            IF (_MessageLevel > E_MessageType.eMessageError)
            THEN
              _stMsg.eType                                    := E_MessageType.eMessageInfo;
              _stMsg.eSubdevice                               := e_Subdevice.Application_Finish;
              _stMsg.iErrorNumber                             := 0;
              _stMsg.sText                                    := concat(TO_STRING(E_INSTANCE.OUTFEED_ROBOT_R1), ': _wDisable ');
              _stMsg.sText                                    := concat(_stMsg.sText, _ItfProcessCollector[E_INSTANCE.OUTFEED_ROBOT_R1].BitsToString(_wDisable));
              f_MessageSet(_stMsg);
            END_IF
          END_IF
        ELSE
          _InstanceCtrl[E_INSTANCE.OUTFEED_ROBOT_R1].Cmd      := E_INSTANCE_CMD.ENABLE;
        END_IF
      END_CASE

      E_INSTANCE_STATE.ENABLED:
        CASE _InstanceState[E_INSTANCE.OUTFEED_ROBOT_R1].Progress
        OF
          E_PROGRESS.PROGRESS_OCCUPIED:
            _InstanceCtrl[E_INSTANCE.OUTFEED_ROBOT_R1].Cmd    := E_INSTANCE_CMD.PROCEED;
        END_CASE


      E_INSTANCE_STATE.WORKING:
        CASE _InstanceState[E_INSTANCE.OUTFEED_ROBOT_R1].Progress
        OF
          E_PROGRESS.PROGRESS_BUSY:
            _tonProcess [E_INSTANCE.OUTFEED_ROBOT_R1]
                                                  (IN         := FALSE, 
                                                   PT         := _tProcess[E_INSTANCE.OUTFEED_ROBOT_R1]);

            _InstanceCtrl[E_INSTANCE.OUTFEED_ROBOT_R1].Cmd    := E_INSTANCE_CMD.WORK;
    

          E_PROGRESS.PROGRESS_CHECK:
            _tonProcess [E_INSTANCE.OUTFEED_ROBOT_R1]
                                                  (IN         := TRUE, 
                                                   PT         := _tProcess[E_INSTANCE.OUTFEED_ROBOT_R1]);
    
            IF _tonProcess [E_INSTANCE.OUTFEED_ROBOT_R1].Q
            THEN
              _InstanceCtrl[E_INSTANCE.OUTFEED_ROBOT_R1].Cmd  := E_INSTANCE_CMD.FINISH;
            END_IF
        END_CASE

      E_INSTANCE_STATE.FINISH:
        CASE _InstanceState[E_INSTANCE.OUTFEED_ROBOT_R1].Progress
        OF
          E_PROGRESS.PROGRESS_BUSY:
            _InstanceCtrl[E_INSTANCE.OUTFEED_ROBOT_R1].Cmd    := E_INSTANCE_CMD.FINISH;

          E_PROGRESS.PROGRESS_DONE:
            _InstanceCtrl[E_INSTANCE.OUTFEED_ROBOT_R1].Cmd    := E_INSTANCE_CMD.DISABLE;
        END_CASE
      END_CASE

    //-------------------------------------------------------------------------
    // E_INSTANCE.OUTFEED_ROBOT_R2
    //-------------------------------------------------------------------------
    CASE _InstanceState[E_INSTANCE.OUTFEED_ROBOT_R2].State
    OF
    E_INSTANCE_STATE.DISABLED:
      CASE _InstanceState[E_INSTANCE.OUTFEED_ROBOT_R2].Progress
      OF
      E_PROGRESS.PROGRESS_BUSY:
        IF (_ItfProcessCollector[E_INSTANCE.OUTFEED_ROBOT_R2].QueueProcessCount < 12)
        THEN
          _InstanceCtrl[E_INSTANCE.OUTFEED_ROBOT_R2].Cmd      := E_INSTANCE_CMD.DISABLE;

          IF NOT (_ItfProcessCollector[E_INSTANCE.OUTFEED_ROBOT_R2].BitGet(_wDisable, TO_BYTE(E_INSTANCE.OUTFEED_ROBOT_R2-1)))
          THEN
            _wDisable                                         := _ItfProcessCollector[E_INSTANCE.OUTFEED_ROBOT_R2].
                                                                 BitSet(_wDisable, TO_BYTE(E_INSTANCE.OUTFEED_ROBOT_R2-1));

            IF (_MessageLevel > E_MessageType.eMessageError)
            THEN
              _stMsg.eType                                    := E_MessageType.eMessageInfo;
              _stMsg.eSubdevice                               := e_Subdevice.Application_Finish;
              _stMsg.iErrorNumber                             := 0;
              _stMsg.sText                                    := concat(TO_STRING(E_INSTANCE.OUTFEED_ROBOT_R2), ': _wDisable ');
              _stMsg.sText                                    := concat(_stMsg.sText, _ItfProcessCollector[E_INSTANCE.OUTFEED_ROBOT_R2].BitsToString(_wDisable));
              f_MessageSet(_stMsg);
            END_IF
          END_IF
        ELSE
          _InstanceCtrl[E_INSTANCE.OUTFEED_ROBOT_R2].Cmd      := E_INSTANCE_CMD.ENABLE;
        END_IF
      END_CASE

      E_INSTANCE_STATE.ENABLED:
        CASE _InstanceState[E_INSTANCE.OUTFEED_ROBOT_R2].Progress
        OF
          E_PROGRESS.PROGRESS_OCCUPIED:
            _InstanceCtrl[E_INSTANCE.OUTFEED_ROBOT_R2].Cmd    := E_INSTANCE_CMD.PROCEED;
        END_CASE

      E_INSTANCE_STATE.WORKING:
        CASE _InstanceState[E_INSTANCE.OUTFEED_ROBOT_R2].Progress
        OF
          E_PROGRESS.PROGRESS_BUSY:
            _tonProcess [E_INSTANCE.OUTFEED_ROBOT_R2]
                                                  (IN         := FALSE, 
                                                   PT         := _tProcess[E_INSTANCE.OUTFEED_ROBOT_R2]);

            _InstanceCtrl[E_INSTANCE.OUTFEED_ROBOT_R2].Cmd    := E_INSTANCE_CMD.WORK;

    
          E_PROGRESS.PROGRESS_CHECK:
            _tonProcess [E_INSTANCE.OUTFEED_ROBOT_R2]
                                                  (IN         := TRUE, 
                                                   PT         := _tProcess[E_INSTANCE.OUTFEED_ROBOT_R2]);
    
            IF _tonProcess [E_INSTANCE.OUTFEED_ROBOT_R2].Q
            THEN
              _InstanceCtrl[E_INSTANCE.OUTFEED_ROBOT_R2].Cmd  := E_INSTANCE_CMD.FINISH;
            END_IF
        END_CASE

      E_INSTANCE_STATE.FINISH:
        CASE _InstanceState[E_INSTANCE.OUTFEED_ROBOT_R2].Progress
        OF
          E_PROGRESS.PROGRESS_BUSY:
            _InstanceCtrl[E_INSTANCE.OUTFEED_ROBOT_R2].Cmd    := E_INSTANCE_CMD.FINISH;

          E_PROGRESS.PROGRESS_DONE:
            _InstanceCtrl[E_INSTANCE.OUTFEED_ROBOT_R2].Cmd    := E_INSTANCE_CMD.DISABLE;
        END_CASE
      END_CASE

    //-------------------------------------------------------------------------
    // E_INSTANCE.SENDER_FAST
    //-------------------------------------------------------------------------
    CASE _InstanceState[E_INSTANCE.SENDER_FAST].State
    OF
      E_INSTANCE_STATE.DISABLED:
        CASE _InstanceState[E_INSTANCE.SENDER_FAST].Progress
        OF
          E_PROGRESS.PROGRESS_BUSY:
            IF NOT (_ItfProcessCollector[E_INSTANCE.OUTFEED_ROBOT_R1].QueueProcessCount < 12) OR 
               NOT (_ItfProcessCollector[E_INSTANCE.OUTFEED_ROBOT_R2].QueueProcessCount < 12)
            THEN
              _InstanceCtrl[E_INSTANCE.SENDER_FAST].Cmd       := E_INSTANCE_CMD.ENABLE;

            ELSIF (_ItfProcessCollector[E_INSTANCE.SENDER_FAST].QueueProcessCount > 0)
            THEN
              _InstanceCtrl[E_INSTANCE.SENDER_FAST].Cmd       := E_INSTANCE_CMD.ENABLE;
            ELSE
              _InstanceCtrl[E_INSTANCE.SENDER_FAST].Cmd       := E_INSTANCE_CMD.DISABLE;

              IF NOT (_ItfProcessCollector[E_INSTANCE.SENDER_FAST].BitGet(_wDisable, TO_BYTE(E_INSTANCE.SENDER_FAST-1)))
              THEN
                _wDisable                                     := _ItfProcessCollector[E_INSTANCE.SENDER_FAST].
                                                                 BitSet(_wDisable, TO_BYTE(E_INSTANCE.SENDER_FAST-1));
    
                IF (_MessageLevel > E_MessageType.eMessageError)
                THEN
                  _stMsg.eType                                := E_MessageType.eMessageInfo;
                  _stMsg.eSubdevice                           := e_Subdevice.Application_Finish;
                  _stMsg.iErrorNumber                         := 0;
                  _stMsg.sText                                := concat(TO_STRING(E_INSTANCE.SENDER_FAST), ': _wDisable ');
                  _stMsg.sText                                := concat(_stMsg.sText, _ItfProcessCollector[E_INSTANCE.SENDER_FAST].BitsToString(_wDisable));
                  f_MessageSet(_stMsg);
                END_IF
              END_IF
            END_IF
        END_CASE

      E_INSTANCE_STATE.FINISH:
        CASE _InstanceState[E_INSTANCE.SENDER_FAST].Progress
        OF
          E_PROGRESS.PROGRESS_BUSY:
            _InstanceCtrl[E_INSTANCE.SENDER_FAST].Cmd         := E_INSTANCE_CMD.FINISH;
        END_CASE
      END_CASE
END_CASE
//-----------------------------------------------------------------------------
//-----------------------------------------------------------------------------
CASE _eState
OF
  E_PROGRESS.PROGRESS_STILL_WORKING:
    _XtsTransportCtrl.Cmd                                 := E_XTS_TRANSPORT_CTRL.CMD_GROUP_STOP;
  
    IF (_XtsTransportState.State = E_XTS_TRANSPORT_STATE.TRANSPORT_GROUP_STOP + E_PROGRESS.PROGRESS_ERROR)
    THEN
      _eState                                             := E_PROGRESS.PROGRESS_ERROR;

      _stMsg.eType                  := E_MessageType.eMessageError;
      _stMsg.eSubdevice             := e_Subdevice.Application_Finish;
      _stMsg.iErrorNumber           := 0;
      _stMsg.sText                  := concat(TO_STRING(_eState), ': ');
      f_MessageSet(_stMsg);

  
    ELSIF (_XtsTransportState.State = E_XTS_TRANSPORT_STATE.TRANSPORT_GROUP_STOP + E_PROGRESS.PROGRESS_DONE)
    THEN
      _eState                                             := E_PROGRESS.PROGRESS_DONE;

      IF (_MessageLevel > E_MessageType.eMessageError)
      THEN
        _stMsg.eType                := E_MessageType.eMessageInfo;
        _stMsg.eSubdevice           := e_Subdevice.Application_Finish;
        _stMsg.iErrorNumber         := 0;
        _stMsg.sText                := concat(TO_STRING(_eState), ': ');
        f_MessageSet(_stMsg);
      END_IF
    END_IF
END_CASE
//-----------------------------------------------------------------------------
//-----------------------------------------------------------------------------

Finish                            := _eState;
END_METHOD

METHOD Init       : E_PROGRESS // used only for first cycle startup, 
                               // use method Clear during operations if you have to clean up the instances 
VAR_INPUT
  Execute         : BOOL;
END_VAR
VAR_INST
  _nIdx,
  _nErrorId       : UDINT;
  _eState         : E_PROGRESS;
END_VAR
//-----------------------------------------------------------------------------
IF NOT Execute 
THEN 
	_eState                                         := E_PROGRESS.PROGRESS_INIT; 
END_IF 
//-----------------------------------------------------------------------------
IF NOT Check() 
THEN 
	Init                                            := E_PROGRESS.PROGRESS_ERROR; 
	RETURN; 
END_IF
//-----------------------------------------------------------------------------
//-----------------------------------------------------------------------------
CASE _eState
OF
  //---------------------------------------------------------------------------------------------------------------
  //---------------------------------------------------------------------------------------------------------------
  E_PROGRESS.PROGRESS_INIT:                   // startup procedure for your application
    IF Execute
    THEN
      _eState                                       := E_PROGRESS.PROGRESS_BUSY;

      IF (_MessageLevel > E_MessageType.eMessageError)
      THEN
        _stMsg.eType            := E_MessageType.eMessageInfo;
        _stMsg.eSubdevice       := e_Subdevice.Application_Init;
        _stMsg.iErrorNumber     := 0;
        _stMsg.sText            := concat(TO_STRING(_eState), ': ');
        f_MessageSet(_stMsg);
      END_IF

      IF (GVL_APPLICATION.bOutput_R1R2)
      THEN
        MAIN_APP.ProcessInit_R1R2();
      ELSE
        MAIN_APP.ProcessInit_CLAMP();
      END_IF

      FOR _nIdx := 1 TO MAX_PROCESS
      DO
        _InstanceCtrl[_nIdx].Cmd                    := E_INSTANCE_CMD.INIT;
      END_FOR
    END_IF
  //---------------------------------------------------------------------------------------------------------------
  //---------------------------------------------------------------------------------------------------------------
  E_PROGRESS.PROGRESS_BUSY:
    _InstanceCtrl[E_INSTANCE.BUFFER_INFEED].Cmd   := E_INSTANCE_CMD.DISABLE;
    //-----------------------------------------------------------------------------------
    CASE _InstanceState[E_INSTANCE.BUFFER_INFEED].State
    OF
      E_INSTANCE_STATE.DISABLED:
        CASE _InstanceState[E_INSTANCE.BUFFER_INFEED].Progress
        OF
          E_PROGRESS.PROGRESS_BUSY:           // check for startup to be done
            _eState                               := E_PROGRESS.PROGRESS_PREPARE; // go check next insatnce
        END_CASE
    END_CASE

  //---------------------------------------------------------------------------------------------------------------
  //---------------------------------------------------------------------------------------------------------------
  E_PROGRESS.PROGRESS_PREPARE:
    _InstanceCtrl[E_INSTANCE.INFEED].Cmd          := E_INSTANCE_CMD.DISABLE;
    //-----------------------------------------------------------------------------------
    CASE _InstanceState[E_INSTANCE.INFEED].State
    OF
      E_INSTANCE_STATE.DISABLED:
        CASE _InstanceState[E_INSTANCE.INFEED].Progress
        OF
          E_PROGRESS.PROGRESS_BUSY:           // check for startup to be done
          _eState                                 := E_PROGRESS.PROGRESS_STARTUP; // go check next insatnce
        END_CASE
    END_CASE

  //---------------------------------------------------------------------------------------------------------------
  //---------------------------------------------------------------------------------------------------------------
  E_PROGRESS.PROGRESS_STARTUP:
    _InstanceCtrl[E_INSTANCE.BUFFER_OUTFEED].Cmd   := E_INSTANCE_CMD.DISABLE;
    //-----------------------------------------------------------------------------------
    CASE _InstanceState[E_INSTANCE.BUFFER_OUTFEED].State
    OF
      E_INSTANCE_STATE.DISABLED:
        CASE _InstanceState[E_INSTANCE.BUFFER_OUTFEED].Progress
        OF
          E_PROGRESS.PROGRESS_BUSY:           // check for startup to be done
          _eState                                 := E_PROGRESS.PROGRESS_CHECK; // go check next insatnce
        END_CASE
    END_CASE

  //---------------------------------------------------------------------------------------------------------------
  //---------------------------------------------------------------------------------------------------------------
  E_PROGRESS.PROGRESS_CHECK:
    _InstanceCtrl[E_INSTANCE.OUTFEED_ROBOT_R1].Cmd   := E_INSTANCE_CMD.DISABLE;
    //-----------------------------------------------------------------------------------
    CASE _InstanceState[E_INSTANCE.OUTFEED_ROBOT_R1].State
    OF
      E_INSTANCE_STATE.DISABLED:
        CASE _InstanceState[E_INSTANCE.OUTFEED_ROBOT_R1].Progress
        OF
          E_PROGRESS.PROGRESS_BUSY:           // check for startup to be done
          _eState                                 := E_PROGRESS.PROGRESS_OCCUPIED; // go check next insatnce
        END_CASE
    END_CASE

  //---------------------------------------------------------------------------------------------------------------
  //---------------------------------------------------------------------------------------------------------------
  E_PROGRESS.PROGRESS_OCCUPIED:
    _InstanceCtrl[E_INSTANCE.OUTFEED_ROBOT_R2].Cmd   := E_INSTANCE_CMD.DISABLE;
    //-----------------------------------------------------------------------------------
    CASE _InstanceState[E_INSTANCE.OUTFEED_ROBOT_R2].State
    OF
      E_INSTANCE_STATE.DISABLED:
        CASE _InstanceState[E_INSTANCE.OUTFEED_ROBOT_R2].Progress
        OF
          E_PROGRESS.PROGRESS_BUSY:           // check for startup to be done
          _eState                                 := E_PROGRESS.PROGRESS_WORKING; // go check next insatnce
        END_CASE
    END_CASE

  //---------------------------------------------------------------------------------------------------------------
  //---------------------------------------------------------------------------------------------------------------
  E_PROGRESS.PROGRESS_WORKING:
    _InstanceCtrl[E_INSTANCE.SENDER_FAST].Cmd     := E_INSTANCE_CMD.DISABLE;
    //-----------------------------------------------------------------------------------
    CASE _InstanceState[E_INSTANCE.SENDER_FAST].State
    OF
      E_INSTANCE_STATE.DISABLED:
        CASE _InstanceState[E_INSTANCE.SENDER_FAST].Progress
        OF
          E_PROGRESS.PROGRESS_BUSY:           // check for startup to be done
          _eState                                 := E_PROGRESS.PROGRESS_STILL_WORKING; // go check next insatnce
        END_CASE
    END_CASE

  //---------------------------------------------------------------------------------------------------------------
  //---------------------------------------------------------------------------------------------------------------
  E_PROGRESS.PROGRESS_STILL_WORKING:
    _InstanceCtrl[E_INSTANCE.SENDER_BUFFER_INFEED].Cmd   := E_INSTANCE_CMD.DISABLE;
    //-----------------------------------------------------------------------------------
    CASE _InstanceState[E_INSTANCE.SENDER_BUFFER_INFEED].State
    OF
      E_INSTANCE_STATE.DISABLED:
        CASE _InstanceState[E_INSTANCE.SENDER_BUFFER_INFEED].Progress
        OF
          E_PROGRESS.PROGRESS_BUSY:           // check for startup to be done
          _eState                                 := E_PROGRESS.PROGRESS_DONE;

          _stMsg.eType                            := E_MessageType.eMessageInfo;
          _stMsg.eSubdevice                       := e_Subdevice.Application_Init;
          _stMsg.iErrorNumber                     := 0;
          _stMsg.sText                            := concat(TO_STRING(_eState), ': ');
          f_MessageSet(_stMsg);
        END_CASE
    END_CASE
END_CASE
//-----------------------------------------------------------------------------
//-----------------------------------------------------------------------------

Init                                              := _eState;
END_METHOD

PROPERTY InstanceCtrl : REFERENCE TO ARRAY[1..MAX_PROCESS] OF ST_INSTANCE_CTRL
SET
_InstanceCtrl REF= InstanceCtrl;
END_SET
END_PROPERTY

PROPERTY InstanceState : REFERENCE TO ARRAY[1..MAX_PROCESS] OF ST_INSTANCE_STATE
SET
_InstanceState REF= InstanceState;
END_SET
END_PROPERTY

METHOD ListData   : E_PROGRESS  // simulates data entry from transfersystem into BUFFER_INFEED linked list
VAR_INPUT
  Start           : BOOL;
  Reset           : BOOL;
END_VAR
VAR_INST
  _nBit,
  _nExp           : BYTE;
  _nMod           : UINT := 5;
  _nCount         : UINT;
  _eStateProgress : E_PROGRESS;

  _ProcessData    : ST_PROCESS_DATA;
  _Rslt           : ST_PROCESS_LIST_RESULT;

  _nMinListCount  : UDINT := 1;
  _nWaitcountLast,
  _nWaitCount     : UDINT;

  _tMsg           : ST_Message;
END_VAR
IF Reset
THEN
  _nCount                     := 1;
  _eStateProgress             := E_PROGRESS.PROGRESS_INIT;
  _ItfProcessList[E_INSTANCE.BUFFER_INFEED].InitList();
END_IF

_tMsg.eDevice                 := _stMsg.eDevice; 

CASE _eStateProgress
OF
   E_PROGRESS.PROGRESS_INIT:
    IF Start
    THEN
      _eStateProgress         :=  E_PROGRESS.PROGRESS_BUSY;
    END_IF

  E_PROGRESS.PROGRESS_BUSY:
    CASE _nLoadCase
    OF
      0:  // fully loaded
        _eStateProgress       := E_PROGRESS.PROGRESS_CHECK;
        _nLoadCaseOld         := _nLoadCase;

        IF (_MessageLevel > E_MessageType.eMessageError)
        THEN
          _tMsg.eType         := E_MessageType.eMessageInfo;
          _tMsg.eSubdevice    := e_Subdevice.Application;
          _tMsg.iErrorNumber  := _nLoadCase;
          _tMsg.sText         := concat('ListData.Progress: ', TO_STRING(_eStateProgress));
          _tMsg.sText         := concat(_tMsg.sText, ': LoadCase: ');
          _tMsg.sText         := concat(_tMsg.sText, TO_STRING(_nLoadCase));
   
          f_MessageSet(_tMsg);
        END_IF


      1:  // static bits
        _eStateProgress       := E_PROGRESS.PROGRESS_PREPARE;
        _nLoadCaseOld         := _nLoadCase;

        IF (_MessageLevel > E_MessageType.eMessageError)
        THEN
          _tMsg.eType          := E_MessageType.eMessageInfo;
          _tMsg.eSubdevice     := e_Subdevice.Application;
          _tMsg.iErrorNumber   := _nLoadCase;
          _tMsg.sText         := concat('ListData.Progress: ', TO_STRING(_eStateProgress));
          _tMsg.sText         := concat(_tMsg.sText, ': LoadCase: ');
          _tMsg.sText         := concat(_tMsg.sText, TO_STRING(_nLoadCase));
          f_MessageSet(_tMsg);
        END_IF


      2:  // incrementing bits
        _eStateProgress       := E_PROGRESS.PROGRESS_STARTUP;
        _nLoadCaseOld         := _nLoadCase;

        IF (_MessageLevel > E_MessageType.eMessageError)
        THEN
          _tMsg.eType          := E_MessageType.eMessageInfo;
          _tMsg.eSubdevice     := e_Subdevice.Application;
          _tMsg.iErrorNumber   := _nLoadCase;
          _tMsg.sText         := concat('ListData.Progress: ', TO_STRING(_eStateProgress));
          _tMsg.sText         := concat(_tMsg.sText, ': LoadCase: ');
          _tMsg.sText         := concat(_tMsg.sText, TO_STRING(_nLoadCase));
          f_MessageSet(_tMsg);
        END_IF


      99:
        _eStateProgress       := E_PROGRESS.PROGRESS_WORKING;
        _ProcessData.wTarget  := 0;

        IF (_MessageLevel > E_MessageType.eMessageError)
        THEN
          _tMsg.eType          := E_MessageType.eMessageInfo;
          _tMsg.eSubdevice     := e_Subdevice.Application;
          _tMsg.iErrorNumber   := _nLoadCase;
          _tMsg.sText          := concat(TO_STRING(_eState), ': _ProcessData.wTarget: ');
          _tMsg.sText          := concat(_stMsg.sText, _ItfProcessCollector[E_INSTANCE.BUFFER_INFEED].BitsToString(_ProcessData.wTarget));
          f_MessageSet(_tMsg);
        END_IF
        _nLoadCase            := _nLoadCaseOld;

    ELSE
        _eStateProgress       := E_PROGRESS.PROGRESS_STARTUP;
    END_CASE
    _nWaitCount               := 0; 
END_CASE
CASE _eStateProgress
OF
  E_PROGRESS.PROGRESS_PREPARE:
    _eStateProgress           := E_PROGRESS.PROGRESS_WORKING;
    _nExp                     := TO_BYTE(ItfProcessCollector[E_INSTANCE.INFEED].StationCount);
    _ProcessData.wTarget      := _ItfProcessCollector[E_INSTANCE.BUFFER_INFEED].To_T_Process(_nExp);

    IF (_nCount MOD _nMod = 0)
    THEN
      _nBit                   := SEL((_nBit>_nExp), _nBit+1, 0);
      _ProcessData.wTarget    := _ItfProcessCollector[E_INSTANCE.BUFFER_INFEED].BitDel(_ProcessData.wTarget, _nBit);
    END_IF
    IF (_nCount MOD (8) = 0)
    THEN
      _nBit                   := 1;
      _ProcessData.wTarget    := _ItfProcessCollector[E_INSTANCE.BUFFER_INFEED].BitDel(_ProcessData.wTarget, _nBit);
    END_IF
    IF (_nCount MOD (16) = 0)
    THEN
      _nBit                   := 2;
      _ProcessData.wTarget    := _ItfProcessCollector[E_INSTANCE.BUFFER_INFEED].BitDel(_ProcessData.wTarget, _nBit);
    END_IF
    IF (_nCount MOD (24) = 0)
    THEN
      _nBit                   := 3;
      _ProcessData.wTarget    := _ItfProcessCollector[E_INSTANCE.BUFFER_INFEED].BitDel(_ProcessData.wTarget, _nBit);
    END_IF
    IF (_nCount MOD (32) = 0)
    THEN
      _nBit                   := 4;
      _ProcessData.wTarget    := _ItfProcessCollector[E_INSTANCE.BUFFER_INFEED].BitDel(_ProcessData.wTarget, _nBit);
    END_IF
    IF (_nCount MOD (40) = 0)
    THEN
      _nBit                   := 5;
      _ProcessData.wTarget    := _ItfProcessCollector[E_INSTANCE.BUFFER_INFEED].BitDel(_ProcessData.wTarget, _nBit);
    END_IF
    IF (_nCount MOD (48) = 0)
    THEN
      _nBit                   := 6;
      _ProcessData.wTarget    := _ItfProcessCollector[E_INSTANCE.BUFFER_INFEED].BitDel(_ProcessData.wTarget, _nBit);
    END_IF
    IF (_nCount MOD (60) = 0)
    THEN
      _nBit                   := 7;
      _ProcessData.wTarget    := _ItfProcessCollector[E_INSTANCE.BUFFER_INFEED].BitDel(_ProcessData.wTarget, _nBit);
    END_IF
    IF (_nCount MOD (72) = 0)
    THEN
      _nBit                   := 8;
      _ProcessData.wTarget    := _ItfProcessCollector[E_INSTANCE.BUFFER_INFEED].BitDel(_ProcessData.wTarget, _nBit);
    END_IF
    IF (_nCount MOD (84) = 0)
    THEN
      _nBit                   := 9;
      _ProcessData.wTarget    := _ItfProcessCollector[E_INSTANCE.BUFFER_INFEED].BitDel(_ProcessData.wTarget, _nBit);
    END_IF
    IF (_nCount MOD (96) = 0)
    THEN
      _nBit                   := 10;
      _ProcessData.wTarget    := _ItfProcessCollector[E_INSTANCE.BUFFER_INFEED].BitDel(_ProcessData.wTarget, _nBit);
    END_IF
    IF (_nCount MOD (108) = 0)
    THEN
      _nBit                   := 11;
      _ProcessData.wTarget    := _ItfProcessCollector[E_INSTANCE.BUFFER_INFEED].BitDel(_ProcessData.wTarget, _nBit);
    END_IF
END_CASE
CASE _eStateProgress
OF
  E_PROGRESS.PROGRESS_STARTUP:
    _eStateProgress           := E_PROGRESS.PROGRESS_WORKING;
    _nExp                     := TO_BYTE(ItfProcessCollector[E_INSTANCE.INFEED].StationCount);
    _ProcessData.wTarget      := _ItfProcessCollector[E_INSTANCE.BUFFER_INFEED].To_T_Process(_nExp);

    IF (_nCount MOD _nMod = 0)
    THEN
      _nBit                   := SEL((_nBit>_nExp), _nBit+1, 0);
      _ProcessData.wTarget    := _ItfProcessCollector[E_INSTANCE.BUFFER_INFEED].BitDel(_ProcessData.wTarget, _nBit);
    END_IF
(*
    IF (_nCount MOD (8) = 0)
    THEN
      _nBit                   := SEL((_nBit>_nExp), _nBit+1, 0);
      _ProcessData.wTarget    := _ItfProcessCollector[E_INSTANCE.BUFFER_INFEED].DelBit(_ProcessData.wTarget, _nBit);
    END_IF
    IF (_nCount MOD (16) = 0)
    THEN
      _nBit                   := SEL((_nBit>_nExp), _nBit+1, 0);
      _ProcessData.wTarget    := _ItfProcessCollector[E_INSTANCE.BUFFER_INFEED].DelBit(_ProcessData.wTarget, _nBit);
    END_IF
    IF (_nCount MOD (24) = 0)
    THEN
      _nBit                   := SEL((_nBit>_nExp), _nBit+1, 0);
      _ProcessData.wTarget    := _ItfProcessCollector[E_INSTANCE.BUFFER_INFEED].DelBit(_ProcessData.wTarget, _nBit);
    END_IF
    IF (_nCount MOD (32) = 0)
    THEN
      _nBit                   := SEL((_nBit>_nExp), _nBit+1, 0);
      _ProcessData.wTarget    := _ItfProcessCollector[E_INSTANCE.BUFFER_INFEED].DelBit(_ProcessData.wTarget, _nBit);
    END_IF
    IF (_nCount MOD (40) = 0)
    THEN
      _nBit                   := SEL((_nBit>_nExp), _nBit+1, 0);
      _ProcessData.wTarget    := _ItfProcessCollector[E_INSTANCE.BUFFER_INFEED].DelBit(_ProcessData.wTarget, _nBit);
    END_IF
    IF (_nCount MOD (48) = 0)
    THEN
      _nBit                   := SEL((_nBit>_nExp), _nBit+1, 0);
      _ProcessData.wTarget    := _ItfProcessCollector[E_INSTANCE.BUFFER_INFEED].DelBit(_ProcessData.wTarget, _nBit);
    END_IF
*)
END_CASE
CASE _eStateProgress
OF
  E_PROGRESS.PROGRESS_CHECK:
    _eStateProgress           := E_PROGRESS.PROGRESS_WORKING;
    _nExp                     := TO_BYTE(ItfProcessCollector[E_INSTANCE.INFEED].StationCount);
    _ProcessData.wTarget      := _ItfProcessCollector[E_INSTANCE.BUFFER_INFEED].To_T_Process(_nExp);

    IF (_MessageLevel > E_MessageType.eMessageError)
    THEN
      _tMsg.eType             := E_MessageType.eMessageInfo;
      _tMsg.eSubdevice        := e_Subdevice.Application;
      _tMsg.iErrorNumber      := _nLoadCase;
      _tMsg.sText             := concat('ListData.Progress: ', TO_STRING(_eState));
      _tMsg.sText             := concat(_tMsg.sText, ': _ProcessData.wTarget: ');
      _tMsg.sText             := concat(_tMsg.sText, _ItfProcessCollector[E_INSTANCE.BUFFER_INFEED].BitsToString(_ProcessData.wTarget));
      f_MessageSet(_tMsg);
    END_IF
    IF (_MessageLevel > E_MessageType.eMessageEmpty)
    THEN
      _tMsg.eType             := E_MessageType.eMessageInfo;
      _tMsg.eDevice           := e_Device.Metrics;
      _tMsg.eSubdevice        := e_Subdevice.Application;
      _tMsg.iErrorNumber      := _nLoadCase;
      _tMsg.sText             := concat('ListData.Progress: ', TO_STRING(_eState));
      _tMsg.sText             := concat(_tMsg.sText, ': _ProcessData.wTarget: ');
      _tMsg.sText             := concat(_tMsg.sText, _ItfProcessCollector[E_INSTANCE.BUFFER_INFEED].BitsToString(_ProcessData.wTarget));
      f_MessageSet(_tMsg);
    END_IF
END_CASE
CASE _eStateProgress
OF
  E_PROGRESS.PROGRESS_WORKING:
    _Rslt                     := _ItfProcessList[E_INSTANCE.BUFFER_INFEED].AddTailValue(_ProcessData);

    IF (_Rslt.wState = 0)
    THEN
      _nCount                 := _nCount + 1;
      _eStateProgress         := E_PROGRESS.PROGRESS_OCCUPIED;
      IF (_MessageLevel > E_MessageType.eMessageError)
      THEN
        _tMsg.eType           := E_MessageType.eMessageInfo;
        _tMsg.eSubdevice      := e_Subdevice.Application;
        _tMsg.iErrorNumber    := _nLoadCase;
        _tMsg.sText           := concat('AddTail: ', TO_STRING(E_INSTANCE.BUFFER_INFEED));
        _tMsg.sText           := concat(_tMsg.sText, ': ');
        _tMsg.sText           := concat(_tMsg.sText, TO_STRING(E_PROGRESS.PROGRESS_DONE));
        f_MessageSet(_tMsg);
      END_IF

    ELSE
      _eStateProgress         := E_PROGRESS.PROGRESS_ERROR;

      IF (_MessageLevel > E_MessageType.eMessageEmpty)
      THEN
        _tMsg.eType           := E_MessageType.eMessageError;
        _tMsg.eSubdevice      := e_Subdevice.Application;
        _tMsg.iErrorNumber    := _nLoadCase;
        _tMsg.sText           := concat('AddTail: ', TO_STRING(E_INSTANCE.BUFFER_INFEED));
        _tMsg.sText           := concat(_tMsg.sText, ': ');
        _tMsg.sText           := concat(_tMsg.sText, TO_STRING(_eStateProgress));
        f_MessageSet(_tMsg);
      END_IF
    END_IF
END_CASE
CASE _eStateProgress
OF
  E_PROGRESS.PROGRESS_OCCUPIED:
    _nWaitCount               := _nWaitCount + 1;

    IF (_ItfProcessList[E_INSTANCE.BUFFER_INFEED].Count < _nMinListCount)
    THEN
      _nWaitCountLast         := _nWaitCount;
      _eStateProgress         :=  E_PROGRESS.PROGRESS_INIT;
    END_IF
END_CASE

ListData                      := _eStateProgress;
END_METHOD

PROPERTY MessageLevel : e_MessageType
GET
MessageLevel := _MessageLevel;
END_GET
SET
_MessageLevel := MessageLevel;
END_SET
END_PROPERTY

METHOD Proceed : E_PROGRESS
VAR_INPUT
  Execute     : BOOL;
END_VAR
VAR_INST
  _nErrorId               : UDINT;
  _eState                 : E_PROGRESS;

  _nExp                   : BYTE;
  _WriteData              : ST_PROCESS_DATA;
  _WriteResult            : ST_PROCESS_LIST_RESULT;

  _eInst                  : E_INSTANCE;
  _TransportState         : E_XTS_TRANSPORT_STATE;
  _bDbg : BOOL;
END_VAR
//-----------------------------------------------------------------------------
IF NOT Execute 
THEN 
	_eState                       := E_PROGRESS.PROGRESS_INIT; 
END_IF 
//-----------------------------------------------------------------------------
IF NOT Check() 
THEN 
	Proceed                       := E_PROGRESS.PROGRESS_ERROR; 
	RETURN; 
END_IF
//-----------------------------------------------------------------------------
//-----------------------------------------------------------------------------
CASE _eState
OF
  E_PROGRESS.PROGRESS_INIT:
    IF Execute
    THEN
      _nErrorId                 := 0;

      IF (_XtsTransportState.GroupInfo.AxisCountEnabled = MAX_MOVER) AND
         (_XtsTransportState.GroupInfo.AxisCount        = MAX_MOVER)
      THEN
        _eState                 := E_PROGRESS.PROGRESS_BUSY;
        _XtsTransportCtrl.Cmd   := E_XTS_TRANSPORT_CTRL.CMD_NULL;

        IF (_MessageLevel > E_MessageType.eMessageError)
        THEN
          _stMsg.eType          := E_MessageType.eMessageInfo;
          _stMsg.eSubdevice     := e_Subdevice.Application_Proceed;
          _stMsg.iErrorNumber   := 0;
          _stMsg.sText          := concat(TO_STRING(_eState), ': ');
          f_MessageSet(_stMsg);
        END_IF
      ELSE
        _nErrorId               := _eState;

        _eState                 := E_PROGRESS.PROGRESS_ERROR;

        _stMsg.eType            := E_MessageType.eMessageError;
        _stMsg.eSubdevice       := e_Subdevice.Application_Proceed;
        _stMsg.iErrorNumber     := _nErrorId;
        _stMsg.sText            := concat(TO_STRING(_eState), ': ');
        _stMsg.sText            := concat(_stMsg.sText, TO_STRING(_XtsTransportState.GroupInfo.AxisCountEnabled));
        _stMsg.sText            := concat(_stMsg.sText, ' / ');
        _stMsg.sText            := concat(_stMsg.sText, TO_STRING(_XtsTransportState.GroupInfo.AxisCount));
        _stMsg.sText            := concat(_stMsg.sText, ' CaGroup Axis mismatch');
        f_MessageSet(_stMsg);
      END_IF
    END_IF


  E_PROGRESS.PROGRESS_BUSY:
    _XtsTransportCtrl.Cmd       := E_XTS_TRANSPORT_CTRL.CMD_TRANSPORT_RESTART;

    IF (_XtsTransportState.State = E_XTS_TRANSPORT_STATE.TRANSPORT_RESTART + E_PROGRESS.PROGRESS_ERROR)
    THEN
      _eState                   := E_PROGRESS.PROGRESS_ERROR;
      _TransportState           := _XtsTransportState.State MOD E_PROGRESS.PROGRESS_ERROR;

      _stMsg.eType              := E_MessageType.eMessageError;
      _stMsg.eSubdevice         := e_Subdevice.Application_Proceed;
      _stMsg.iErrorNumber       := _nErrorId;
      _stMsg.sText              := concat(TO_STRING(_eState), ': ');
      _stMsg.sText              := concat(_stMsg.sText, TO_STRING(_TransportState));
      f_MessageSet(_stMsg);

    ELSIF (_XtsTransportState.State = E_XTS_TRANSPORT_STATE.TRANSPORT_RESTART + E_PROGRESS.PROGRESS_DONE)
    THEN
      _eState                   := E_PROGRESS.PROGRESS_WORKING;
      _TransportState           := _XtsTransportState.State MOD E_PROGRESS.PROGRESS_DONE;

      IF (_MessageLevel > E_MessageType.eMessageError)
      THEN
        _stMsg.eType            := E_MessageType.eMessageInfo;
        _stMsg.eSubdevice       := e_Subdevice.Application_Proceed;
        _stMsg.iErrorNumber     := 0;
        _stMsg.sText            := concat(TO_STRING(_eState), ': ');
        _stMsg.sText            := concat(_stMsg.sText, TO_STRING(_TransportState));
        f_MessageSet(_stMsg);
      END_IF
    END_IF

END_CASE
//-----------------------------------------------------------------------------
//-----------------------------------------------------------------------------
CASE _eState
OF
  E_PROGRESS.PROGRESS_WORKING:
    ListData(TRUE, FALSE);    // start writing linked list entries into BUFFER_INFEED

    FOR _eInst := E_INSTANCE.BUFFER_INFEED TO E_INSTANCE.SENDER_BUFFER_INFEED
    DO
      // handshakes to instances: 
      // - deconstruct this for your own implementation
      CASE _InstanceState[_eInst].State
      OF
        E_INSTANCE_STATE.DISABLED:
          CASE _InstanceState[_eInst].Progress
          OF
            E_PROGRESS.PROGRESS_BUSY:
              _InstanceCtrl[_eInst].Cmd    := E_INSTANCE_CMD.ENABLE;
          END_CASE
      
        E_INSTANCE_STATE.ENABLED:
          CASE _InstanceState[_eInst].Progress
          OF
            E_PROGRESS.PROGRESS_OCCUPIED:
              _InstanceCtrl[_eInst].Cmd    := E_INSTANCE_CMD.PROCEED;
          END_CASE
      
        E_INSTANCE_STATE.WORKING:
          CASE _InstanceState[_eInst].Progress
          OF
            E_PROGRESS.PROGRESS_BUSY:
              _tonProcess [_eInst]
                              (IN         := FALSE, 
                               PT         := _tProcess[_eInst]);

              IF (_eInst > E_INSTANCE.OUTFEED_ROBOT_R2) OR
                 (_eInst < E_INSTANCE.OUTFEED_ROBOT_R1) OR
                 (_bSingleOutput) OR
                 NOT (GVL_APPLICATION.bOutput_R1R2)
              THEN
                _InstanceCtrl[_eInst].Cmd   := E_INSTANCE_CMD.WORK;
              ELSE
                IF (_InstanceState[E_INSTANCE.OUTFEED_ROBOT_R1].State = 
                    _InstanceState[E_INSTANCE.OUTFEED_ROBOT_R2].State )
                THEN
                  // in this example the outfeed instances are working in sync
                  _InstanceCtrl[_eInst].Cmd := E_INSTANCE_CMD.WORK;
                ELSE
                  CASE _InstanceState[E_INSTANCE.OUTFEED_ROBOT_R2].State
                  OF
                    E_INSTANCE_STATE.ENABLED:
                      // in case R2 is empty --> unload R1
                      _InstanceCtrl[E_INSTANCE.OUTFEED_ROBOT_R1].Cmd := E_INSTANCE_CMD.WORK;
                  END_CASE
                END_IF
              END_IF
      
      
            E_PROGRESS.PROGRESS_CHECK:
              _tonProcess [_eInst]
                              (IN         := TRUE, 
                               PT         := _tProcess[_eInst]);
      
              IF _tonProcess [_eInst].Q
              THEN
                _InstanceCtrl[_eInst].Cmd := E_INSTANCE_CMD.FINISH;
              END_IF
          END_CASE


        E_INSTANCE_STATE.FINISH:
          CASE _InstanceState[_eInst].Progress
          OF
            E_PROGRESS.PROGRESS_BUSY:
              _InstanceCtrl[_eInst].Cmd    := E_INSTANCE_CMD.FINISH;

            E_PROGRESS.PROGRESS_OCCUPIED:
              _InstanceCtrl[_eInst].Cmd    := E_INSTANCE_CMD.PROCEED;
          END_CASE
        END_CASE
    END_FOR
END_CASE
//-----------------------------------------------------------------------------
//-----------------------------------------------------------------------------

Proceed                            := _eState;
END_METHOD

PROPERTY ProcessLinkedLists : REFERENCE TO ARRAY[1..MAX_PROCESS] OF I_Process_LinkedList
SET
_ItfProcessList REF= ProcessLinkedLists;
END_SET
END_PROPERTY

PROPERTY State : REFERENCE TO ST_APP_STATE
SET
_State ref= State;
END_SET
END_PROPERTY

METHOD Work : E_PROGRESS  // cyclic handshakes with timers, 
                          // this procedure you have to build for your own application. 
                          // This simulated work method is here 
                          // because it was convinient for me to do so
VAR_INPUT
  Execute                 : BOOL;
END_VAR
VAR_INST
  _nErrorId               : UDINT;
  _eRslt,
  _eState                 : E_PROGRESS;

  _nExp                   : BYTE;
  _WriteData              : ST_PROCESS_DATA;
  _WriteResult            : ST_PROCESS_LIST_RESULT;

  _eInst                  : E_INSTANCE;
  _bDbg : BOOL;

  _TransportState         : E_XTS_TRANSPORT_STATE;
  _JobResult              : E_PROGRESS;
END_VAR
//-----------------------------------------------------------------------------
IF NOT Execute 
THEN 
	_eState                       := E_PROGRESS.PROGRESS_INIT; 
END_IF 
//-----------------------------------------------------------------------------
IF NOT Check() 
THEN 
	Work                          := E_PROGRESS.PROGRESS_ERROR; 
	RETURN; 
END_IF
//-----------------------------------------------------------------------------
//-----------------------------------------------------------------------------
CASE _eState
OF
  E_PROGRESS.PROGRESS_INIT:
    IF Execute
    THEN
      IF (GVL_APPLICATION.bOutput_R1R2)
      THEN
        MAIN_APP.ProcessInit_R1R2();
  
        _stMsg.eType                             := E_MessageType.eMessageInfo;
        _stMsg.eSubdevice                        := e_Subdevice.Application_Work;
        _stMsg.iErrorNumber                      := _eState;
        _stMsg.sText                             := concat('Application.Work: ', TO_STRING(_eState));
        _stMsg.sText                             := concat(_stMsg.sText, ': ');
        _stMsg.sText                             := concat(_stMsg.sText, TO_STRING(E_INSTANCE.OUTFEED_ROBOT_R1));
        _stMsg.sText                             := concat(_stMsg.sText, ': ');
        _stMsg.sText                             := concat(_stMsg.sText, TO_STRING(E_INSTANCE.OUTFEED_ROBOT_R2));
        f_MessageSet(_stMsg);
      ELSE
  
        MAIN_APP.ProcessInit_CLAMP();

        _stMsg.eType                             := E_MessageType.eMessageInfo;
        _stMsg.eSubdevice                        := e_Subdevice.Application_Work;
        _stMsg.iErrorNumber                      := _eState;
        _stMsg.sText                             := concat('Application.Work: ', TO_STRING(_eState));
        _stMsg.sText                             := concat(_stMsg.sText, ': ');
        _stMsg.sText                             := concat(_stMsg.sText, TO_STRING(E_INSTANCE.OUTFEED_ROBOT_R1));
        f_MessageSet(_stMsg);
      END_IF

      _nErrorId                 := 0;

      IF (_XtsTransportState.GroupInfo.AxisCountEnabled = MAX_MOVER) AND
         (_XtsTransportState.GroupInfo.AxisCount        = MAX_MOVER)
      THEN
        _eState                 := E_PROGRESS.PROGRESS_BUSY;
        _XtsTransportCtrl.Cmd   := E_XTS_TRANSPORT_CTRL.CMD_NULL;
        _eRslt                  := Clear(FALSE);

        IF (_MessageLevel > E_MessageType.eMessageError)
        THEN
          _stMsg.eType          := E_MessageType.eMessageInfo;
          _stMsg.eSubdevice     := e_Subdevice.Application_Work;
          _stMsg.iErrorNumber   := 0;
          _stMsg.sText          := concat(TO_STRING(_eState), ': ');
          f_MessageSet(_stMsg);
        END_IF
      ELSE
        _nErrorId               := _XtsTransportState.GroupInfo.AxisCountEnabled;
        _eState                 := E_PROGRESS.PROGRESS_ERROR;

        _stMsg.eType            := E_MessageType.eMessageError;
        _stMsg.eSubdevice       := e_Subdevice.Application_Work;
        _stMsg.iErrorNumber     := _nErrorId;
        _stMsg.sText            := concat(TO_STRING(_eState), ': ');
        _stMsg.sText            := concat(_stMsg.sText, TO_STRING(_XtsTransportState.GroupInfo.AxisCountEnabled));
        _stMsg.sText            := concat(_stMsg.sText, ' / ');
        _stMsg.sText            := concat(_stMsg.sText, TO_STRING(_XtsTransportState.GroupInfo.AxisCount));
        _stMsg.sText            := concat(_stMsg.sText, ' CaGroup Axis mismatch');
        f_MessageSet(_stMsg);
      END_IF
    END_IF


  E_PROGRESS.PROGRESS_BUSY:
    _eRslt                      := Clear(TRUE);

    IF (_eRslt = E_PROGRESS.PROGRESS_DONE)
    THEN
      _XtsTransportCtrl.Cmd     := E_XTS_TRANSPORT_CTRL.CMD_TRANSPORT_START;
  
      IF (_XtsTransportState.State = E_XTS_TRANSPORT_STATE.TRANSPORT_START + E_PROGRESS.PROGRESS_ERROR)
      THEN
        _eState                 := E_PROGRESS.PROGRESS_ERROR;
        _TransportState         := _XtsTransportState.State MOD E_PROGRESS.PROGRESS_ERROR;

        _stMsg.eType            := E_MessageType.eMessageError;
        _stMsg.eSubdevice       := e_Subdevice.Application_Work;
        _stMsg.iErrorNumber     := _nErrorId;
        _stMsg.sText            := concat(TO_STRING(_eState), ': ');
        _stMsg.sText            := concat(_stMsg.sText, TO_STRING(_TransportState));
        f_MessageSet(_stMsg);
  
      ELSIF (_XtsTransportState.State = E_XTS_TRANSPORT_STATE.TRANSPORT_START + E_PROGRESS.PROGRESS_DONE)
      THEN
        _eState                 := E_PROGRESS.PROGRESS_PREPARE;
        _TransportState         := _XtsTransportState.State MOD E_PROGRESS.PROGRESS_DONE;

        IF (_MessageLevel > E_MessageType.eMessageError)
        THEN
          _stMsg.eType          := E_MessageType.eMessageInfo;
          _stMsg.eSubdevice     := e_Subdevice.Application_Work;
          _stMsg.iErrorNumber   := 0;
          _stMsg.sText          := concat(TO_STRING(_eState), ': ');
          _stMsg.sText          := concat(_stMsg.sText, TO_STRING(_TransportState));
          f_MessageSet(_stMsg);
        END_IF
      END_IF
    END_IF
END_CASE
//-----------------------------------------------------------------------------
//-----------------------------------------------------------------------------
CASE _eState
OF
  E_PROGRESS.PROGRESS_PREPARE:  // SENDER_BUFFER_INFEED sends the first batch of movers to BUFFER_INFEED
                                //  - after sending the first batch 
                                //    --> the transfersystem (ListData) may start writing entries into BUFFER_INFEED
    CASE _InstanceState[E_INSTANCE.SENDER_BUFFER_INFEED].State
    OF
    E_INSTANCE_STATE.DISABLED:

      CASE _InstanceState[E_INSTANCE.SENDER_BUFFER_INFEED].Progress
      OF
      E_PROGRESS.PROGRESS_BUSY:
        _nExp                   := TO_BYTE(ItfProcessCollector[E_INSTANCE.INFEED].StationCount);
        _WriteData.wTarget      := _ItfProcessCollector[E_INSTANCE.SENDER_BUFFER_INFEED].To_T_Process(_nExp);

        _WriteResult            := _ItfProcessList[E_INSTANCE.SENDER_BUFFER_INFEED].AddTailValue(_WriteData);

        IF (_WriteResult.wState <> 0)
        THEN
          _eState               := E_PROGRESS.PROGRESS_ERROR;

          _stMsg.eType          := E_MessageType.eMessageError;
          _stMsg.eSubdevice     := e_Subdevice.Application_Work;
          _stMsg.iErrorNumber   := _WriteResult.wState;
          _stMsg.sText          := concat(TO_STRING(_eState), ': ');
          _stMsg.sText          := concat(_stMsg.sText, TO_STRING(e_Subdevice.Process_LinkedList_AddTail));
          f_MessageSet(_stMsg);

        ELSE
          ListData(FALSE, TRUE);    // init linked list from simulated transfersystem (timer based entry into linked list)
          _eState               := E_PROGRESS.PROGRESS_CHECK;

          IF (_MessageLevel > E_MessageType.eMessageError)
          THEN
            _stMsg.eType        := E_MessageType.eMessageInfo;
            _stMsg.eSubdevice   := e_Subdevice.Application_Work;
            _stMsg.iErrorNumber := 0;
            _stMsg.sText        := concat(TO_STRING(_eState), ': ');
            _stMsg.sText        := concat(_stMsg.sText, TO_STRING(e_Subdevice.Process_LinkedList_AddTail));
            f_MessageSet(_stMsg);
          END_IF
        END_IF
      END_CASE
    END_CASE
END_CASE
//-----------------------------------------------------------------------------
//-----------------------------------------------------------------------------
CASE _eState
OF
  E_PROGRESS.PROGRESS_CHECK:
    _eState := E_PROGRESS.PROGRESS_OCCUPIED; 
END_CASE
//-----------------------------------------------------------------------------
//-----------------------------------------------------------------------------
CASE _eState
OF
  E_PROGRESS.PROGRESS_OCCUPIED:
    _eState := E_PROGRESS.PROGRESS_WORKING;

    IF (_MessageLevel > E_MessageType.eMessageError)
    THEN
      _stMsg.eType            := E_MessageType.eMessageInfo;
      _stMsg.eSubdevice       := e_Subdevice.Application_Work;
      _stMsg.iErrorNumber     := 0;
      _stMsg.sText            := concat(TO_STRING(_eState), ': ');
      f_MessageSet(_stMsg);
    END_IF
END_CASE
//-----------------------------------------------------------------------------
//-----------------------------------------------------------------------------
CASE _eState
OF
  E_PROGRESS.PROGRESS_WORKING:
    ListData(TRUE, FALSE);    // start writing linked list entries into BUFFER_INFEED

    FOR _eInst := E_INSTANCE.BUFFER_INFEED TO E_INSTANCE.SENDER_BUFFER_INFEED
    DO
      // handshakes to instances: 
      // - deconstruct this for your own implementation
      CASE _InstanceState[_eInst].State
      OF
        E_INSTANCE_STATE.DISABLED:
          CASE _InstanceState[_eInst].Progress
          OF
            E_PROGRESS.PROGRESS_BUSY:
              _InstanceCtrl[_eInst].Cmd    := E_INSTANCE_CMD.ENABLE;
          END_CASE
      
        E_INSTANCE_STATE.ENABLED:
          CASE _InstanceState[_eInst].Progress
          OF
            E_PROGRESS.PROGRESS_OCCUPIED:
              _InstanceCtrl[_eInst].Cmd    := E_INSTANCE_CMD.PROCEED;
          END_CASE

        E_INSTANCE_STATE.WORKING:
          CASE _InstanceState[_eInst].Progress
          OF
            E_PROGRESS.PROGRESS_BUSY:
              _tonProcess [_eInst]
                              (IN         := FALSE, 
                               PT         := _tProcess[_eInst]);


              IF (_eInst > E_INSTANCE.OUTFEED_ROBOT_R2) OR
                 (_eInst < E_INSTANCE.OUTFEED_ROBOT_R1) OR
                 (_bSingleOutput) OR
                 NOT (GVL_APPLICATION.bOutput_R1R2)
              THEN
                _InstanceCtrl[_eInst].Cmd   := E_INSTANCE_CMD.WORK;
              ELSE
                IF (_InstanceState[E_INSTANCE.OUTFEED_ROBOT_R1].State = 
                    _InstanceState[E_INSTANCE.OUTFEED_ROBOT_R2].State )
                THEN
                  // in this example the outfeed instances are working in sync
                  _InstanceCtrl[_eInst].Cmd := E_INSTANCE_CMD.WORK;
                END_IF
              END_IF
      
      
            E_PROGRESS.PROGRESS_CHECK:
              _tonProcess [_eInst]
                              (IN         := TRUE, 
                               PT         := _tProcess[_eInst]);
      
              IF _tonProcess [_eInst].Q
              THEN
                _InstanceCtrl[_eInst].Cmd := E_INSTANCE_CMD.FINISH;
              END_IF
          END_CASE


        E_INSTANCE_STATE.FINISH:
          CASE _InstanceState[_eInst].Progress
          OF
            E_PROGRESS.PROGRESS_BUSY:
              _tonProcess [_eInst]
                              (IN         := FALSE, 
                               PT         := _tProcess[_eInst]);

              _InstanceCtrl[_eInst].Cmd    := E_INSTANCE_CMD.FINISH;

            E_PROGRESS.PROGRESS_OCCUPIED:
              _InstanceCtrl[_eInst].Cmd    := E_INSTANCE_CMD.PROCEED;
          END_CASE
        END_CASE
    END_FOR
END_CASE
//-----------------------------------------------------------------------------
//-----------------------------------------------------------------------------

Work                            := _eState;
END_METHOD

PROPERTY WriteTimeVariant : bool
GET
WriteTimeVariant := _bWriteTimeVariant;
END_GET
SET
_bWriteTimeVariant := WriteTimeVariant;
END_SET
END_PROPERTY

PROPERTY XtsTransportCtrl : REFERENCE TO ST_XTS_TRANSPORT_CTRL
SET
_XtsTransportCtrl REF= XtsTransportCtrl;
END_SET
END_PROPERTY

PROPERTY XtsTransportState : REFERENCE TO ST_XTS_TRANSPORT_STATE
SET
_XtsTransportState REF= XtsTransportState;
END_SET
END_PROPERTY

END_FUNCTION_BLOCK

// ---- APPLICATION/Process_Instances/fb_BufferInfeed.TcPOU
//---------------------------------------------------------------------------------------------------------------
//
//  HAUD 2024.11.15
//
//
//  fb_BufferInfeed
//  - inherits fb_Instance, which provides a design pattern in order to build different specific processes in a structured way
//  - uses a single XtsStation via _ItfProcessCollector
//  - used for targeting movers to predetermined substations of process control (1 to many)
//  - processes are connected via linked list
//    - entry in list is detected
//    - entry in list determines count and place of used XtsStations in target process
//
//
//  - constructed with fb_Instance main state (_eStateInstance) in addition to a substate (_eStateProgress)
//  - substate enables to handle procedures within main state by preventing race conditions 
//    with the help of small steps and decisions with clear separation from each other 
//
//---------------------------------------------------------------------------------------------------------------//
// This SOFTWARE is provided as an Exemple by THE PROVIDER "as is" and "with all faults." THE PROVIDER makes no  //
// representations or warranties of any kind concerning the safety, suitability, lack of viruses, inaccuracies,  //
// typographical errors, or other harmful components of this SOFTWARE. There are inherent dangers in the use of  //
// any software, and you are solely responsible for determining whether this SOFTWARE is compatible with your    //
// equipment and other software installed on your equipment. You are also solely responsible for the protection  //
// of your equipment and backup of your data, and THE PROVIDER will not be liable for any damages you may suffer //
// in connection with using, modifying, or distributing this SOFTWARE.                                           //
//---------------------------------------------------------------------------------------------------------------//
FUNCTION_BLOCK fb_BufferInfeed EXTENDS fb_Instance
VAR
  _nProcessTarget               : E_INSTANCE;     // who am I connected to

  // target XTS station range
  _nTargetStationLast           : UINT;           // where does the target process end
  _nTargetStationFirst          : UINT;           // where does the target process start

  _rCheckPos                    : LREAL;

  _WriteResult                  : ST_PROCESS_LIST_RESULT;   // last job written to target
  _DeleteResult                 : ST_PROCESS_LIST_RESULT;   // last job executed

  _idx                          : UINT;
  _nTargetIndex                 : ARRAY[1..SIZEOF(T_PROCESS)*8] OF USINT;

  _MoverInfo                    : ST_MOVER_INFO;      // Information from the Mover in Station
  _StationState                 : ST_STATION_STATE;   // BufferInfeed has only one XtsStation to work
END_VAR

//-----------------------------------------------------------------------------
//-----------------------------------------------------------------------------
// check pointer and interface
// connect Ctrl/State to _ItfProcessCollector
// set message device identification
//-----------------------------------------------------------------------------
IF NOT Check() THEN 
  RETURN; 
END_IF
//-----------------------------------------------------------------------------
// check command
//-----------------------------------------------------------------------------
_eCmd                                 := _InstanceCtrl[_nProcess].Cmd;
IF (_eCmd <> _eCmdOld)
THEN
  CASE _eCmd
  OF
    E_INSTANCE_CMD.INIT:
      // clear init info
      _eInit                          := _ItfProcessCollector[_nProcess].Init(FALSE);
  
      IF _ItfProcessList[_nProcess].InitList()  // clear linked list
      THEN
        Clear();
        _eStateInstance               := E_INSTANCE_STATE.INIT;
        _eStateProgress               := E_PROGRESS.PROGRESS_INIT;
      END_IF
  END_CASE
  CmdLog();
  _eCmdOld                            := _eCmd;
END_IF

//-----------------------------------------------------------------------------
//-----------------------------------------------------------------------------
// state machine for BufferInfeed work
//-----------------------------------------------------------------------------
CASE _eStateInstance
OF
  E_INSTANCE_STATE.NULL:
    // first cycle startup
    // initialize linked list, clears all entries
    IF _ItfProcessList[_nProcess].InitList()
    THEN
      _eInit                          := _ItfProcessCollector[_nProcess].Init(FALSE);
      _eStateProgress                 := E_PROGRESS.PROGRESS_INIT;
      _eStateInstance                 := E_INSTANCE_STATE.INIT;
    END_IF


  E_INSTANCE_STATE.INIT:
    //-------------------------------------------------------------------------
    CASE _eStateProgress
    OF
    // E_INSTANCE_STATE.INIT:
    //-------------------------------------------------------------------------
      E_PROGRESS.PROGRESS_ERROR:
        IF (_nProcessTarget > 0) AND
           (_nProcessTarget < E_INSTANCE.INSTANCE_MAX)
        THEN
          _eStateProgress             := E_PROGRESS.PROGRESS_INIT;
        END_IF

    // E_INSTANCE_STATE.INIT:
    //-------------------------------------------------------------------------
      E_PROGRESS.PROGRESS_INIT:
        IF NOT (_nProcessTarget > 0) OR
           NOT (_nProcessTarget < E_INSTANCE.INSTANCE_MAX)
        THEN
          _eStateProgress             := E_PROGRESS.PROGRESS_ERROR;

        ELSE
          _eStateProgress             := E_PROGRESS.PROGRESS_BUSY;
        END_IF

    // E_INSTANCE_STATE.INIT:
    //-------------------------------------------------------------------------
      E_PROGRESS.PROGRESS_BUSY:
        // wait for process collector check to be done
        //  - checks range of XtsStations
        //  - checks count of XtsStations
        IF (_State.Check = E_PROCESS_CHECK.PROCESS_CHECK_DONE)
        THEN
          _eInit                      := _ItfProcessCollector[_nProcess].Init(TRUE);
  
          IF (_eInit = E_PROGRESS.PROGRESS_DONE)
          THEN
            IF NOT (_nProcessTarget > 0) OR
               NOT (_nProcessTarget < E_INSTANCE.INSTANCE_MAX)
            THEN
              // an invalid target you must have not
              _eStateProgress         := E_PROGRESS.PROGRESS_ERROR;

              _stMsg.eType            := E_MessageType.eMessageError;
              _stMsg.eSubdevice       := e_Subdevice.Instance_BufferInfeed;
              _stMsg.iErrorNumber     := _nProcessTarget;
              _stMsg.sText            := concat(TO_STRING(_eStateInstance), ': ProcessTarget: ');
              _stMsg.sText            := concat(_stMsg.sText, TO_STRING(_eStateProgress));
              f_MessageSet(_stMsg);

            ELSE
              _ItfProcessCollector[_nProcess].Init(FALSE); // clear init procedure

              // for ease of use; copy target XtsStation range to local helper vars
              _nTargetStationLast     := _ItfProcessCollector[_nProcessTarget].StationLast;
              _nTargetStationFirst    := _ItfProcessCollector[_nProcessTarget].StationFirst;
      
              // initialization of BufferInfeed: _ItfProcessCollector with XtsStation
              _Ctrl.Cmd               := E_PROCESS_CTRL.PROCESS_DISABLE;  // switch off _ItfProcessCollector and XtsStation
              _eStateProgress         := E_PROGRESS.PROGRESS_INIT;        // clear sub state
              _eStateInstance         := E_INSTANCE_STATE.DISABLED;       // switch to disabled as default after startup
            END_IF
          END_IF
        END_IF
    END_CASE
END_CASE
//-----------------------------------------------------------------------------
// DISABLED:
//  - clear local list result data
//  - wait for enable from the outside
//-----------------------------------------------------------------------------
CASE _eStateInstance
OF
  E_INSTANCE_STATE.DISABLED:
    //-------------------------------------------------------------------------
    CASE _eStateProgress
    OF
      E_PROGRESS.PROGRESS_INIT:
        _Ctrl.Cmd                     := E_PROCESS_CTRL.PROCESS_DISABLE;  // switch off _ItfProcessCollector and XtsStation
        _eStateProgress               := E_PROGRESS.PROGRESS_BUSY;
        // clear data for a new round
        memset(ADR(_ListResult), 0, SIZEOF(_ListResult));

        _Ctrl.ActivateStation         := 0; // clear activation mask of my process
        _Ctrl.NestMask                := 1; // my process target has one nest
    END_CASE
    // E_INSTANCE_STATE.DISABLED:
    //-------------------------------------------------------------------------
    CASE _eStateProgress
    OF
      E_PROGRESS.PROGRESS_BUSY:
        CASE _eCmd
        OF
          E_INSTANCE_CMD.ENABLE:      // turn it on!!
            _eStateInstance           := E_INSTANCE_STATE.DETECTION;
            _eStateProgress           := E_PROGRESS.PROGRESS_BUSY;
  
            IF (_MessageLevel > E_MessageType.eMessageInfo)
            THEN
              _stMsg.eType            := E_MessageType.eMessageVerbose;
              _stMsg.eSubdevice       := e_Subdevice.Instance_BufferInfeed;
              _stMsg.iErrorNumber     := 0;
              _stMsg.sText            := concat(TO_STRING(_eStateInstance), ': ');
              _stMsg.sText            := concat(_stMsg.sText, TO_STRING(_eStateProgress));
              f_MessageSet(_stMsg);
            END_IF

        END_CASE
    END_CASE
END_CASE
//-----------------------------------------------------------------------------
// DETECTION: 
//  - check inked list and GetHead()
//  - copy job data
//  - switch on process
//-----------------------------------------------------------------------------
CASE _eStateInstance
OF
  E_INSTANCE_STATE.DETECTION:
    //-------------------------------------------------------------------------
    CASE _eStateProgress
    OF
      E_PROGRESS.PROGRESS_INIT:
        IF (_eCmd = E_INSTANCE_CMD.PROCEED)
        THEN
          _eStateProgress             := E_PROGRESS.PROGRESS_BUSY;
        END_IF
    END_CASE
    // E_INSTANCE_STATE.DETECTION
    //-------------------------------------------------------------------------
    CASE _eStateProgress
    OF
      E_PROGRESS.PROGRESS_BUSY:
        IF (_eCmd = E_INSTANCE_CMD.DISABLE)
        THEN
          _eStateInstance             := E_INSTANCE_STATE.DISABLED;
          _eStateProgress             := E_PROGRESS.PROGRESS_INIT;

        ELSIF (_ItfProcessList[_nProcess].Count > 0)
        THEN
          // get new job order for my process
          // check my list for a new round of movers
          _ListResult                 := _ItfProcessList[_nProcess].GetHead();  // the list results carries information about the requirements of the target process (who and where)

          IF (_ListResult.wState <> 0)
          THEN
            // error in list results must not appear
            // if you land here, there is somethng wrong with the initialization or configuration of the linked list
            _eStateProgress           := E_PROGRESS.PROGRESS_ERROR;

            _stMsg.eType              := E_MessageType.eMessageError;
            _stMsg.eSubdevice         := e_Subdevice.Process_LinkedList_GetHead;
            _stMsg.iErrorNumber       := _ListResult.wState;
            _stMsg.sText              := concat(TO_STRING(_eStateInstance), ': _ListResult.wState: ');
            _stMsg.sText              := concat(_stMsg.sText, TO_STRING(_eStateProgress));
            f_MessageSet(_stMsg);

          ELSE
            IF (_MessageLevel > E_MessageType.eMessageError)
            THEN
              _stMsg.eType            := E_MessageType.eMessageInfo;
              _stMsg.eSubdevice       := e_Subdevice.Process_LinkedList_GetHead;
              _stMsg.iErrorNumber     := 0;
              _stMsg.sText            := concat(TO_STRING(_eStateInstance), ': ');
              _stMsg.sText            := concat(_stMsg.sText, '_ListResult.stData.wTarget: ');
              _stMsg.sText            := concat(_stMsg.sText, _ItfProcessCollector[_nProcess].BitsToString(_ListResult.stData.wTarget));
              f_MessageSet(_stMsg);
            END_IF

            _ProcessData              := _ListResult.stData;  // list result contains data for target process

            IF (_ProcessData.wTarget > 0)
            THEN
              _eStateProgress         := E_PROGRESS.PROGRESS_CHECK;

              IF (_MessageLevel > E_MessageType.eMessageEmpty)
              THEN
                _stMsg.eType          := E_MessageType.eMessageBatch;
                _stMsg.eSubdevice     := e_Subdevice.Instance_BufferInfeed;
                _stMsg.iErrorNumber   := 0;
                _stMsg.sText          := concat(TO_STRING(_eStateProgress), ': ');
                _stMsg.sText          := concat(_stMsg.sText, TO_STRING(e_message_batch.MSG_BATCH_JOB_STARTED));
                f_MessageSet(_stMsg);
              END_IF
            ELSE
              _DeleteResult           := _ItfProcessList[_nProcess].RemoveHeadValue();
            END_IF

            // check target mask for entries
            IF NOT (_ProcessData.wTarget > 0)
            THEN
              //_eStateProgress         := E_PROGRESS.PROGRESS_ERROR;

              _stMsg.eType            := E_MessageType.eMessageWarning;
              _stMsg.eSubdevice       := e_Subdevice.Process_LinkedList_CheckData;
              _stMsg.iErrorNumber     := 666;
              _stMsg.sText            := concat(TO_STRING(_eStateInstance), ': ');
              _stMsg.sText            := concat(_stMsg.sText, '_ProcessData.wTarget: ');
              _stMsg.sText            := concat(_stMsg.sText, _ItfProcessCollector[_nProcess].BitsToString(_ProcessData.wTarget));
              f_MessageSet(_stMsg);
            END_IF
          END_IF
        END_IF
    END_CASE
    // E_INSTANCE_STATE.DETECT_IN_LIST
    //-------------------------------------------------------------------------
    CASE _eStateProgress
    OF
      E_PROGRESS.PROGRESS_CHECK:
        // check for disabled process interface state
        CASE _State.State
        OF
          E_PROCESS_STATE.PROCESS_DISABLE:

          CASE _State.Result
          OF
            E_PROGRESS.PROGRESS_BUSY:     // busy from _State.Result means, waiting for input
              // now the preparation for the target process may begin
              _Ctrl.Cmd               := E_PROCESS_CTRL.PROCESS_ENABLE; // switch on my state machine in _ItfProcessCollector
              _Ctrl.ActivateStation   := 1;                             // enable my XtsStation in _ItfProcessCollector (BufferInfeed has only one XtsStation)

              _eStateInstance         := E_INSTANCE_STATE.ENABLED;      // go check if my process is switched on
              _eStateProgress         := E_PROGRESS.PROGRESS_INIT;      // reset substate

              IF (_MessageLevel > E_MessageType.eMessageInfo)
              THEN
                _stMsg.eType          := E_MessageType.eMessageVerbose;
                _stMsg.eSubdevice     := e_Subdevice.Instance_BufferInfeed;
                _stMsg.iErrorNumber   := 0;
                _stMsg.sText          := concat(TO_STRING(_eStateInstance), ': ');
                _stMsg.sText          := concat(_stMsg.sText, TO_STRING(_eStateProgress));
                _stMsg.sText          := concat(_stMsg.sText, ': ');
                _stMsg.sText          := concat(_stMsg.sText, TO_STRING(_Ctrl.Cmd));
                f_MessageSet(_stMsg);
              END_IF
          END_CASE
        END_CASE
    END_CASE
END_CASE
//-----------------------------------------------------------------------------
// ENABLED
//  - check process for enabled stations from list entry
//  - switch to infeed
//  - check if infeed is active on all required stations
//  - allow movers to enter
//  - check if movers arrived at PosStop[1]
//-----------------------------------------------------------------------------
CASE _eStateInstance
OF
  E_INSTANCE_STATE.ENABLED:
    //-------------------------------------------------------------------------
    CASE _eStateProgress
    OF
      E_PROGRESS.PROGRESS_INIT:
        CASE _State.State
        OF
          E_PROCESS_STATE.PROCESS_ENABLE:
          CASE _State.Result
          OF
            E_PROGRESS.PROGRESS_BUSY:
              // now my process and all XtsStations within are switched on
              // check infeed into my process
              _Ctrl.Cmd               := E_PROCESS_CTRL.PROCESS_STATIONS_INFEED; // tells my process to go check the infeed
              _eStateProgress         := E_PROGRESS.PROGRESS_BUSY; // go check how the infeed into my process is doing

              _StationState           := _ItfProcessCollector[_nProcess].GetStationState  (_ItfProcessCollector[_nProcess].StationLast);
              _MoverInfo              := _ItfProcessCollector[_nProcess].GetMoverInStation(_ItfProcessCollector[_nProcess].StationLast);


              IF (_MessageLevel > E_MessageType.eMessageWarning)
              THEN
                _stMsg.eType          := E_MessageType.eMessageInfo;
                _stMsg.eSubdevice     := e_Subdevice.Instance_BufferInfeed;
                _stMsg.iErrorNumber   := _StationState.nMoverId;
                _stMsg.sText          := concat(TO_STRING(_eStateInstance), ': ');
                _stMsg.sText          := concat(_stMsg.sText, TO_STRING(_eStateProgress));
                _stMsg.sText          := concat(_stMsg.sText, ': ');
                _stMsg.sText          := concat(_stMsg.sText, TO_STRING(_Ctrl.Cmd));
                f_MessageSet(_stMsg);
              END_IF
          END_CASE
        END_CASE
    END_CASE
    // E_INSTANCE_STATE.ENABLED:
    //-------------------------------------------------------------------------
    CASE _eStateProgress
    OF
      E_PROGRESS.PROGRESS_BUSY:
        CASE _State.State
        OF
          E_PROCESS_STATE.PROCESS_STATIONS_INFEED:
          CASE _State.Result
          OF
            E_PROGRESS.PROGRESS_INIT:
              CASE _eCmd
              OF
                E_INSTANCE_CMD.DISABLE:
                  _eStateInstance     := E_INSTANCE_STATE.DISABLED;
                  _eStateProgress     := E_PROGRESS.PROGRESS_INIT;
              END_CASE

            E_PROGRESS.PROGRESS_BUSY:
              _StationState           := _ItfProcessCollector[_nProcess].GetStationState  (_ItfProcessCollector[_nProcess].StationLast);
              _MoverInfo              := _ItfProcessCollector[_nProcess].GetMoverInStation(_ItfProcessCollector[_nProcess].StationLast);

            IF TRUE or (_MoverInfo.rModuloActPos < GVL_XTS.StationParameter[53].rPosWait + 50.0) 
              // this 'smaller than' makes sense here because this Process is right behind the modulo turn, 
              // so every mover smaller than the wait position is close enough to start processing
              // why so 'dirty'?    
              //  - I have not abstracted it further 
              //      because this is intended to be the highest Layer 
              //        of transportation and I thought it may have some explicitness in it, 
              //          the fb_Application part will be your job 
              //            when integrating this approach into your world.
            THEN
              // now we know who wants to enter
              _Ctrl.Cmd               := E_PROCESS_CTRL.PROCESS_STATIONS_SEND; // the InfeedBuffer does not need a standstill at PosStop, --> send mover at once

              _eStateInstance         := E_INSTANCE_STATE.FINISH;   // go get data ready for outfeed
              _eStateProgress         := E_PROGRESS.PROGRESS_INIT;  // reset substate

              IF (_MessageLevel > E_MessageType.eMessageError)
              THEN
                _stMsg.eType          := E_MessageType.eMessageInfo;
                _stMsg.eSubdevice     := e_Subdevice.Instance_BufferInfeed;
                _stMsg.iErrorNumber   := _StationState.nMoverId;
                _stMsg.sText          := concat(TO_STRING(_eStateInstance), ': ');
                _stMsg.sText          := concat(_stMsg.sText, TO_STRING(_eStateProgress));
                _stMsg.sText          := concat(_stMsg.sText, ': ');
                _stMsg.sText          := concat(_stMsg.sText, TO_STRING(_Ctrl.Cmd));
                f_MessageSet(_stMsg);
              END_IF
            END_IF
          END_CASE
        END_CASE
    END_CASE
END_CASE
//-----------------------------------------------------------------------------
// FINISH:
//  - write target (Infeed: Last to First)
//  - delete target bit from linked list result (_ProcessData.wTarget)
//  - send out mover
//  - check _ProcessData.wTarget for next mover
//  - check if all movers in job were sent (ProcessData.wTarget = 0)
//  - RemoveHead() from my list
//  - AddTail() at TargetProcess
//  - check to proceed
//-----------------------------------------------------------------------------
CASE _eStateInstance
OF
  E_INSTANCE_STATE.FINISH:
    //-------------------------------------------------------------------------
    CASE _eStateProgress
    OF
      E_PROGRESS.PROGRESS_INIT:
      // check bit mask for sending mover to required targets
      // get target index for mover from process list entry
      FOR _idx := _nTargetStationLast TO _nTargetStationFirst BY(-1)
      DO
        IF (ItfProcessCollector[_nProcess].BitGet(_ProcessData.wTarget, _idx-_nTargetStationFirst))
        THEN
          _eStateProgress             := E_PROGRESS.PROGRESS_BUSY;

          _nTargetIndex[1]                            := TO_USINT(_idx);
          _ItfProcessCollector[_nProcess].TargetIndex := _nTargetIndex; // write Xts target onto my ProcessCollector interface

          IF (_MessageLevel > E_MessageType.eMessageVerbose)
          THEN
            _stMsg.eType              := E_MessageType.eMessageSentient;
            _stMsg.eSubdevice         := e_Subdevice.Instance_BufferInfeed;
            _stMsg.iErrorNumber       := _idx;
            _stMsg.sText              := concat('I_AM _ProcessData.wTarget: ', 
                                         _ItfProcessCollector[_nProcess].BitsToString(_ProcessData.wTarget));
            f_MessageSet(_stMsg);
          END_IF

          // got the target, now delete the just found bit of this job
          _ProcessData.wTarget        := _ItfProcessCollector[_nProcess].
                                         BitDel(_ProcessData.wTarget, _idx-_nTargetStationFirst);

          IF (_MessageLevel > E_MessageType.eMessageVerbose)
          THEN
            _stMsg.eType              := E_MessageType.eMessageSentient;
            _stMsg.eSubdevice         := e_Subdevice.Instance_BufferInfeed;
            _stMsg.iErrorNumber       := _idx;
            _stMsg.sText              := concat('I_WAS _ProcessData.wTarget: ', 
                                         _ItfProcessCollector[_nProcess].BitsToString(_ProcessData.wTarget));
            f_MessageSet(_stMsg);
          END_IF
          EXIT;
        END_IF
      END_FOR
    END_CASE
    // E_INSTANCE_STATE.FINISH:
    //-------------------------------------------------------------------------
    CASE _eStateProgress
    OF
      E_PROGRESS.PROGRESS_BUSY:
        CASE _State.State
        OF
          E_PROCESS_STATE.PROCESS_STATIONS_OUTFEED: // double check my process' state
          CASE _State.Result
          OF
            E_PROGRESS.PROGRESS_BUSY:
              // now data is prepared and copied to the right places
              _Ctrl.Cmd               := E_PROCESS_CTRL.PROCESS_STATIONS_OUTFEED; // tell my process to release the mover
              _eStateProgress         := E_PROGRESS.PROGRESS_CHECK; // go check for more to do

              IF (_MessageLevel = E_MessageType.eMessageVerbose)
              THEN
                _stMsg.eType          := E_MessageType.eMessageVerbose;
                _stMsg.eSubdevice     := e_Subdevice.Instance_BufferInfeed;
                _stMsg.iErrorNumber   := 0;
                _stMsg.sText          := concat(TO_STRING(_eStateInstance), ': ');
                _stMsg.sText          := concat(_stMsg.sText, TO_STRING(_eStateProgress));
                _stMsg.sText          := concat(_stMsg.sText, ': ');
                _stMsg.sText          := concat(_stMsg.sText, TO_STRING(_Ctrl.Cmd));
                f_MessageSet(_stMsg);
              END_IF
          END_CASE
        END_CASE
    END_CASE
    // E_INSTANCE_STATE.FINISH:
    //-------------------------------------------------------------------------
    CASE _eStateProgress
    OF
      E_PROGRESS.PROGRESS_CHECK:
        CASE _State.State
        OF
          E_PROCESS_STATE.PROCESS_DISABLE:
            IF (_ProcessData.wTarget <> 0)
            THEN
              //_eStateProgress         := E_PROGRESS.PROGRESS_OCCUPIED;
              _Ctrl.Cmd               := E_PROCESS_CTRL.PROCESS_ENABLE; // switch on my state machine in _ItfProcessCollector
              _Ctrl.ActivateStation   := 1;                             // enable my XtsStation in _ItfProcessCollector (BufferInfeed has only one XtsStation)

              _eStateInstance         := E_INSTANCE_STATE.ENABLED;      // go check if my process is switched on
              _eStateProgress         := E_PROGRESS.PROGRESS_INIT;      // reset substate

              IF (_MessageLevel > E_MessageType.eMessageEmpty)
              THEN
                _stMsg.eType          := E_MessageType.eMessageBatch;
                _stMsg.eSubdevice     := e_Subdevice.Instance_BufferInfeed;
                _stMsg.iErrorNumber   := 0;
                _stMsg.sText          := concat(TO_STRING(_eStateProgress), ': ');
                _stMsg.sText          := concat(_stMsg.sText, TO_STRING(e_message_batch.MSG_BATCH_NEXT_IN_JOB));
                f_MessageSet(_stMsg);
              END_IF
              IF (_MessageLevel > E_MessageType.eMessageVerbose)
              THEN
                _stMsg.eType              := E_MessageType.eMessageSentient;
                _stMsg.eSubdevice         := e_Subdevice.Instance_BufferInfeed;
                _stMsg.iErrorNumber       := 0;
                _stMsg.sText              := concat('I_RETURN _ProcessData.wTarget: ', 
                                             _ItfProcessCollector[_nProcess].BitsToString(_ProcessData.wTarget));
                f_MessageSet(_stMsg);
              END_IF
            ELSE
              // job done, all movers were sent
              // job done, delete from top of my list
              _DeleteResult           := _ItfProcessList[_nProcess].RemoveHeadValue();

              IF (_DeleteResult.wState <> 0)
              THEN
                // deleting from list must be successful
                // IF you land here, there is something wrong with initialization or configuration of the linked list
                _eStateProgress       := E_PROGRESS.PROGRESS_ERROR;
              ELSE
                _eStateProgress       := E_PROGRESS.PROGRESS_WORKING; // job is done, now go and write ticket to _nTargetProcess
              END_IF
            END_IF 
        END_CASE
    END_CASE
    // E_INSTANCE_STATE.FINISH:
    //-------------------------------------------------------------------------
    CASE _eStateProgress
    OF
      E_PROGRESS.PROGRESS_OCCUPIED:
        IF (_eCmd = E_INSTANCE_CMD.PROCEED)
        THEN
          // job not finished, go back and get next mover
          _eStateInstance             := E_INSTANCE_STATE.DETECTION;
          _eStateProgress             := E_PROGRESS.PROGRESS_CHECK;
        END_IF
    END_CASE
    // E_INSTANCE_STATE.FINISH:
    //-------------------------------------------------------------------------
    CASE _eStateProgress
    OF
      E_PROGRESS.PROGRESS_WORKING:
        // write process ticket, then go back up
        _WriteResult                  := _ItfProcessList[_nProcessTarget].AddTailValue(_ListResult.stData);

        IF (_WriteResult.wState <> 0)
        THEN
          // adding to target list must be successful on the first try
          // IF you land here, there is something wrong with initialization or configuration of the linked list
          _eStateProgress             := E_PROGRESS.PROGRESS_ERROR;
        ELSE
          _eStateProgress             := E_PROGRESS.PROGRESS_DONE;

          IF (_MessageLevel > E_MessageType.eMessageVerbose)
          THEN
            _stMsg.eType              := E_MessageType.eMessageSentient;
            _stMsg.eSubdevice         := e_Subdevice.Instance_BufferInfeed;
            _stMsg.iErrorNumber       := 0;
            _stMsg.sText              := concat('I_GONE _ProcessData.wTarget: ', 
                                         _ItfProcessCollector[_nProcess].BitsToString(_ProcessData.wTarget));
            f_MessageSet(_stMsg);
          END_IF
          IF (_MessageLevel > E_MessageType.eMessageError)
          THEN
            _stMsg.eType              := E_MessageType.eMessageInfo;
            _stMsg.eSubdevice         := e_Subdevice.Process_LinkedList_AddTail;
            _stMsg.iErrorNumber       := _nProcessTarget;
            _stMsg.sText              := concat(TO_STRING(_eStateInstance), ': ');
            _stMsg.sText              := concat(_stMsg.sText, TO_STRING(_eStateProgress));
            f_MessageSet(_stMsg);
          END_IF
          IF (_MessageLevel > E_MessageType.eMessageEmpty)
          THEN
            _stMsg.eType              := E_MessageType.eMessageBatch;
            _stMsg.eSubdevice         := e_Subdevice.Instance_BufferInfeed;
            _stMsg.iErrorNumber       := 0;
            _stMsg.sText              := concat(TO_STRING(_eStateProgress), ': ');
            _stMsg.sText              := concat(_stMsg.sText, TO_STRING(e_message_batch.MSG_BATCH_JOB_DONE));
            f_MessageSet(_stMsg);
          END_IF
        END_IF
    END_CASE
    // E_INSTANCE_STATE.FINISH:
    //-------------------------------------------------------------------------
    CASE _eStateProgress
    OF
      E_PROGRESS.PROGRESS_DONE:
        _eStateInstance               := E_INSTANCE_STATE.DISABLED;
        _eStateProgress               := E_PROGRESS.PROGRESS_INIT;
    END_CASE
END_CASE
//-----------------------------------------------------------------------------
//-----------------------------------------------------------------------------
_InstanceState[_nProcess].State       := _eStateInstance;
_InstanceState[_nProcess].Progress    := _eStateProgress;

PROPERTY CheckPosition : lreal
GET
CheckPosition := _rCheckPos;
END_GET
SET
_rCheckPos := CheckPosition;
END_SET
END_PROPERTY

METHOD Clear : BOOL
VAR_INPUT
END_VAR
memset(ADR(_nTargetIndex), 0, SIZEOF(_nTargetIndex));

//_eStateInstance                         := E_INSTANCE_STATE.DISABLED;
_eStateProgress                 := E_PROGRESS.PROGRESS_INIT;

Clear                           := TRUE;
END_METHOD

PROPERTY ProcessTarget : E_INSTANCE
GET
ProcessTarget := _nProcessTarget;
END_GET
SET
_nProcessTarget := ProcessTarget;
END_SET
END_PROPERTY

END_FUNCTION_BLOCK

// ---- APPLICATION/_types/Instance/fb_Instance.TcPOU
//---------------------------------------------------------------------------------------------------------------
//
//  HAUD 2024.11.21
//
//
//  fb_Instance
//-----------------------------------------------------------------------------
//  - base class for my process instance to work with fb_ProcessCollector
//
//  - _nProcess --> whoami, this is me
//
//  - fb_ProcessCollector[_nProcess].Cycle() is called in APPLICATION(PRG)
//    - handles range of XtsStations
//    - range must be closed and in consecutive order
//
//    - combines states into bitmasks, one bit per XtsStation
//    - controls forwarding of commands to range of XtsStations 
//      (see fb_ProcessCollector.Cycle())
//
//  - reference to all _ItfProcessCollector(I_ProcessCollector)[]
//    - _ItfProcessCollector[nProcess] Get/Set properties and methods
//
//  - Control / State of my process
//    - datafield for control and state provided
//    - _Ctrl 
//      --> commands to my process; fb_ProcessCollector[_nProcess]
//      --> is linked (REF=) automatically in Check()
//
//      Cmd               : E_PROCESS_CTRL; // command enum for my process
//      ProcessTarget     : UINT;           // target of my process
//      ActivateStation   : WORD;           // is checked for every job
//                                          // every bit is a XtsStation
//
//      NestMask          : BYTE;           // one mask for all XtsStations
//      - every bit is a PosStop in a XtsStation
//      - copied to every XtsStation in my process when movers are about to leave
//
//    - _State
//      --> satus information from my process
//      --> check for plausible StationLast / StationFirst range of XtsStations
//
//      State             : E_PROCESS_STATE;  // state enuum from my process
//      Result            : E_PROGRESS;       // substate from my process, BUSY signals state is ready for interaction
//      Check             : E_PROCESS_CHECK;  // plausibility check of StationLast and StationFirst 
//
//
//  - basic check and var names, so you can build your procedures with it
//
//  - processes may be connected via linked list, you decide.
//    - linked list for processes is intended to work as job buffer
//    - linked list provides information via ST_PROCESS_DATA, 
//      add what you have to in there
//    - linked ist to all process instances provided
//
//  - inherit this base class for your application, call Check() cyclic
//
//---------------------------------------------------------------------------------------------------------------//
// This SOFTWARE is provided as an Exemple by THE PROVIDER "as is" and "with all faults." THE PROVIDER makes no  //
// representations or warranties of any kind concerning the safety, suitability, lack of viruses, inaccuracies,  //
// typographical errors, or other harmful components of this SOFTWARE. There are inherent dangers in the use of  //
// any software, and you are solely responsible for determining whether this SOFTWARE is compatible with your    //
// equipment and other software installed on your equipment. You are also solely responsible for the protection  //
// of your equipment and backup of your data, and THE PROVIDER will not be liable for any damages you may suffer //
// in connection with using, modifying, or distributing this SOFTWARE.                                           //
//---------------------------------------------------------------------------------------------------------------//
FUNCTION_BLOCK ABSTRACT fb_Instance
VAR
  // process index
  _nProcess               : E_INSTANCE;           // whoami

  _InstanceCtrl           : REFERENCE TO ARRAY[1..MAX_PROCESS] OF ST_INSTANCE_CTRL;
  _InstanceState          : REFERENCE TO ARRAY[1..MAX_PROCESS] OF ST_INSTANCE_STATE;

  _eCmd,
  _eCmdOld                : E_INSTANCE_CMD;       // commands for local state machine
  _eStateInstance         : E_INSTANCE_STATE;     // local state machine for infeed procedure

  _eResult,
  _eStateProgress         : E_PROGRESS;           // substate for lacal state machine

  _eInit                  : E_PROGRESS;           // startup
  _eCheck                 : E_INSTANCE_CHECK;     // pointer checks


  // local ctrl / state datafields for you to use, connected by reference to _ItfProcessCollector[_nProcess]
  _Ctrl                   : ST_PROCESS_CTRL;      // control to write, connected by reference to _ItfProcessCollector
  _State                  : ST_PROCESS_STATE;     // state   to read,  connected by reference to _ItfProcessCollector

  _ItfProcessCollector    : ARRAY[1..MAX_PROCESS] OF I_ProcessCollector;    // information and configuration of the connected ProcessCollector for given range of XtsStations

  _ItfProcessList         : ARRAY[1..MAX_PROCESS] OF I_Process_LinkedList;  // access to all linked lists for process entry
  _ListResult             : ST_PROCESS_LIST_RESULT;
  _ProcessData            : ST_PROCESS_DATA;

  {attribute 'displaymode':='bin'}
  _wTargetMask            : ARRAY[1..SIZEOF(T_PROCESS)*8] OF BYTE; // bits for PosStop[] to use in XtsStation of target process

  _stMsg                  : ST_Message;
  _MessageLevel           : E_MessageType;
END_VAR

METHOD Check : BOOL // call this method in the extending/inheriting class
//-----------------------------------------------------------------------------
//-----------------------------------------------------------------------------
// plausibility checks
//-----------------------------------------------------------------------------
IF NOT (_nProcess > 0)
THEN
  _eCheck                 := E_INSTANCE_CHECK.INVALID_PROCESS_ID_ZERO;
  RETURN;
END_IF

IF NOT (_nProcess < E_INSTANCE.INSTANCE_MAX)
THEN
  _eCheck                 := E_INSTANCE_CHECK.INVALID_PROCESS_ID_MAX;
  RETURN;
END_IF
//-----------------------------------------------------------------------------
//-----------------------------------------------------------------------------
// pointer checks
//-----------------------------------------------------------------------------
IF NOT __ISVALIDREF(_InstanceCtrl)
THEN
  _eCheck                 := E_INSTANCE_CHECK.INVALID_INSTANCE_CONTROL_REFERENCE;
  RETURN;
END_IF

IF NOT __ISVALIDREF(_InstanceState)
THEN
  _eCheck                 := E_INSTANCE_CHECK.INVALID_INSTANCE_STATE_REFERENCE;
  RETURN;
END_IF

IF NOT (_ItfProcessCollector[_nProcess] <> 0) 
THEN
  _eCheck                 := E_INSTANCE_CHECK.INVALID_INTERFACE_POINTER;
  RETURN;
END_IF

IF NOT (_ItfProcessCollector[_nProcess].ProcessId > 0)
THEN
  _eCheck                 := E_INSTANCE_CHECK.INVALID_PROCESS_ID_ZERO;
  RETURN;
END_IF

IF NOT (_ItfProcessCollector[_nProcess].ProcessId < E_INSTANCE.INSTANCE_MAX)
THEN
  _eCheck                 := E_INSTANCE_CHECK.INVALID_PROCESS_ID_MAX;
  RETURN;
END_IF

IF NOT (_nProcess = _ItfProcessCollector[_nProcess].ProcessId)
THEN
  _eCheck                 := E_INSTANCE_CHECK.INVALID_PROCESS_ID_NOTEQUAL_COLLECTOR_ID;
  RETURN;
END_IF

IF NOT (_ItfProcessList[_nProcess] <> 0)
THEN
  _eCheck                 := E_INSTANCE_CHECK.INVALID_INDEX_IN_LIST;
  RETURN;
END_IF
//-----------------------------------------------------------------------------
//-----------------------------------------------------------------------------
// connect datafields to interface of ProcessCollector
//-----------------------------------------------------------------------------
_ItfProcessCollector[_nProcess].ProcessCtrl   REF= _Ctrl;
_ItfProcessCollector[_nProcess].ProcessState  REF= _State;

//-----------------------------------------------------------------------------
//-----------------------------------------------------------------------------
// set message device
//-----------------------------------------------------------------------------
_stMsg.eDevice            := e_Device.Process + TO_UINT(_nProcess);
//-----------------------------------------------------------------------------
//-----------------------------------------------------------------------------
_eCheck                   := E_INSTANCE_CHECK.CHECK_DONE;
Check                     := TRUE;
END_METHOD

METHOD CmdLog

IF (_MessageLevel > E_MessageType.eMessageError)
THEN
  _stMsg.eSubdevice       := e_Subdevice.Instance_Command;
  _stMsg.iErrorNumber     := _nProcess;
  _stMsg.sText            := concat('E_INSTANCE_CMD', '.');
  _stMsg.sText            := concat(_stMsg.sText, TO_STRING(_eCmd));
  f_MessageSet(_stMsg);
END_IF
END_METHOD

PROPERTY CollectorInterface : array[1..MAX_PROCESS] of I_ProcessCollector
SET
_ItfProcessCollector := CollectorInterface;
END_SET
END_PROPERTY

PROPERTY InstanceCtrl : REFERENCE TO ARRAY[1..MAX_PROCESS] OF ST_INSTANCE_CTRL
SET
_InstanceCtrl ref= InstanceCtrl;
END_SET
END_PROPERTY

PROPERTY InstanceState : REFERENCE TO ARRAY[1..MAX_PROCESS] OF ST_INSTANCE_STATE
SET
_InstanceState ref= InstanceState;
END_SET
END_PROPERTY

PROPERTY MessageLevel : e_MessageType
GET
MessageLevel := _MessageLevel;
END_GET
SET
_MessageLevel := MessageLevel;

IF NOT (_eInit  = E_PROGRESS.PROGRESS_DONE) OR
   NOT (_eCheck = E_INSTANCE_CHECK.CHECK_DONE)
THEN
  RETURN;
ELSE
  _ItfProcessCollector[_nProcess].MessageLevel := _MessageLevel;
END_IF
END_SET
END_PROPERTY

PROPERTY ProcessId : E_INSTANCE
GET
ProcessId := _nProcess;
END_GET
SET
_nProcess := ProcessId;
END_SET
END_PROPERTY

PROPERTY ProcessLinkedLists : ARRAY[1..max_process] OF I_Process_LinkedList
SET
_ItfProcessList := ProcessLinkedLists;
END_SET
END_PROPERTY

END_FUNCTION_BLOCK

// ---- APPLICATION/Process_Instances/fb_BufferOutfeed.TcPOU
//---------------------------------------------------------------------------------------------------------------
//
//  HAUD 2025.02.20
//
//
//  fb_BufferOutfeedRobot
//  - inherits fb_Instance, which provides a design pattern in order to build different specific processes in a structured way
//  - uses 1 XtsStation via _ItfProcessCollector
//  - used for targeting movers to predetermined substation of process control (one to many)
//  - process checks queue for new movers
//
//
//  - constructed with fb_Instance main state (_eState) in addition to a substate (_eStateProgress)
//  - substate enables to handle procedures within main state by preventing race conditions 
//    with the help of small steps and decisions with clear separation from each other 
//
//---------------------------------------------------------------------------------------------------------------//
// This SOFTWARE is provided as an Exemple by THE PROVIDER "as is" and "with all faults." THE PROVIDER makes no  //
// representations or warranties of any kind concerning the safety, suitability, lack of viruses, inaccuracies,  //
// typographical errors, or other harmful components of this SOFTWARE. There are inherent dangers in the use of  //
// any software, and you are solely responsible for determining whether this SOFTWARE is compatible with your    //
// equipment and other software installed on your equipment. You are also solely responsible for the protection  //
// of your equipment and backup of your data, and THE PROVIDER will not be liable for any damages you may suffer //
// in connection with using, modifying, or distributing this SOFTWARE.                                           //
//---------------------------------------------------------------------------------------------------------------//
FUNCTION_BLOCK fb_BufferOutfeed EXTENDS fb_Instance
VAR
  _nProcessTarget               : ARRAY[1..2] OF E_INSTANCE;     // who am I connected to: OutputR1 and OutputR2

  // target XTS station range
  _nTargetStationLast           : ARRAY[1..2] OF UINT;           // where does the target process end
  _nTargetStationFirst          : ARRAY[1..2] OF UINT;           // where does the target process start

  _rCheckPos                    : LREAL;

  _WriteResult                  : ST_PROCESS_LIST_RESULT;   // last job written to target
  _DeleteResult                 : ST_PROCESS_LIST_RESULT;   // last job executed

  _idx                          : UINT;
  _nTargetIndex                 : ARRAY[1..SIZEOF(T_PROCESS)*8] OF USINT; // helper var to copy to my process (_ItfProcessCollector[_nProcess].TargetIndex)

  _nTargetTotal,                          // how many XtsStations do the target processes have
  _nTargetCounter               : BYTE;   // decremented after every mover, initialized on E_INSTANCE_CMD.INIT

  _MoverInfo                    : ST_MOVER_INFO;      // Information from the Mover in Station
  _StationState                 : ST_STATION_STATE;   // fb_BufferOutfeedRobot has only one XtsStation to work
END_VAR

//-----------------------------------------------------------------------------
//-----------------------------------------------------------------------------
// check pointer and interface
// connect Ctrl/State to _ItfProcessCollector
// set message device identification
//-----------------------------------------------------------------------------
IF NOT Check() THEN 
  RETURN; 
END_IF
//-----------------------------------------------------------------------------
// check init command (hard reset)
//-----------------------------------------------------------------------------
_eCmd                                 := _InstanceCtrl[_nProcess].Cmd;
IF (_eCmd <> _eCmdOld)
THEN
  CASE _eCmd
  OF
    E_INSTANCE_CMD.INIT:
      // clear init info
      _eInit                          := _ItfProcessCollector[_nProcess].Init(FALSE);
  
      IF _ItfProcessList[_nProcess].InitList()  // clear linked list
      THEN
        Clear();
        _eStateInstance               := E_INSTANCE_STATE.INIT;
        _eStateProgress               := E_PROGRESS.PROGRESS_INIT;
      END_IF
  END_CASE
  CmdLog();
  _eCmdOld                            := _eCmd;
END_IF
//-----------------------------------------------------------------------------
// cyclic information of mover and station
//-----------------------------------------------------------------------------
_StationState                         := _ItfProcessCollector[_nProcess].GetStationState  (_ItfProcessCollector[_nProcess].StationLast);
_MoverInfo                            := _ItfProcessCollector[_nProcess].GetMoverInStation(_ItfProcessCollector[_nProcess].StationLast);
//-----------------------------------------------------------------------------
//-----------------------------------------------------------------------------
// state machine for buffer to OutputR1 and OutputR2
//-----------------------------------------------------------------------------
CASE _eStateInstance // main state machine
OF
  E_INSTANCE_STATE.NULL:           // first cycle init
    IF _ItfProcessList[_nProcess].InitList()
    THEN
      _eInit                          := _ItfProcessCollector[_nProcess].Init(FALSE);
      _eStateProgress                 := E_PROGRESS.PROGRESS_INIT;
      _eStateInstance                 := E_INSTANCE_STATE.INIT;
    END_IF


  E_INSTANCE_STATE.INIT:              // plausibility checks and _ItfProcessCollector Init
    //-------------------------------------------------------------------------
    CASE _eStateProgress
    OF
    //-------------------------------------------------------------------------
      E_PROGRESS.PROGRESS_ERROR:
        IF (_nProcessTarget[1] > 0) AND
           (_nProcessTarget[1] < E_INSTANCE.INSTANCE_MAX)
        THEN
          IF (_nProcessTarget[2] > 0) AND
             (_nProcessTarget[2] < E_INSTANCE.INSTANCE_MAX)
          THEN
            _eStateProgress           := E_PROGRESS.PROGRESS_INIT;
          END_IF
        END_IF

    // E_INSTANCE_STATE.INIT:
    //-------------------------------------------------------------------------
      E_PROGRESS.PROGRESS_INIT:
        IF NOT (_nProcessTarget[1] > 0) OR
           NOT (_nProcessTarget[1] < E_INSTANCE.INSTANCE_MAX)
        THEN
          // an invalid target you must have not
          _eStateProgress             := E_PROGRESS.PROGRESS_ERROR;
        ELSE
          IF NOT (_nProcessTarget[2] > 0) OR
             NOT (_nProcessTarget[2] < E_INSTANCE.INSTANCE_MAX)
          THEN
            // an invalid target you must have not
            _eStateProgress           := E_PROGRESS.PROGRESS_ERROR;
          ELSE
            _eStateProgress           := E_PROGRESS.PROGRESS_BUSY;
          END_IF
        END_IF

    // E_INSTANCE_STATE.INIT:
    //-------------------------------------------------------------------------
      E_PROGRESS.PROGRESS_BUSY:
        // wait for my process collector check (_State.Check) to be done
        //  - checks range of XtsStations
        //  - checks count of XtsStations
        IF (_State.Check = E_PROCESS_CHECK.PROCESS_CHECK_DONE)
        THEN
          _eInit                      := _ItfProcessCollector[_nProcess].Init(TRUE);
  
          IF (_eInit = E_PROGRESS.PROGRESS_DONE)
          THEN
            IF NOT (_nProcessTarget[1] > 0) OR
               NOT (_nProcessTarget[1] < E_INSTANCE.INSTANCE_MAX)
            THEN
              // an invalid target you must have not
              _eStateProgress         := E_PROGRESS.PROGRESS_ERROR;
            ELSE
              IF NOT (_nProcessTarget[2] > 0) OR
                 NOT (_nProcessTarget[2] < E_INSTANCE.INSTANCE_MAX)
              THEN
                // an invalid target you must have not
                _eStateProgress       := E_PROGRESS.PROGRESS_ERROR;
              ELSE
                FOR _idx := 1 TO 2
                DO 
                  _nTargetStationLast [_idx]  := _ItfProcessCollector[_nProcessTarget[_idx]].StationLast;
                  _nTargetStationFirst[_idx]  := _ItfProcessCollector[_nProcessTarget[_idx]].StationFirst;
                END_FOR
                // get total of xts stations to serve
                _nTargetTotal         := TO_BYTE(_nTargetStationLast [2] - _nTargetStationFirst[1] + 1);
                // init target counter
                _nTargetCounter       := 0;

